LIN {X 0,Y 250.299,Z 339.512,A -85,B 0,C 180,E1 -19332.01,E2 -19332.01} C_VEL
LIN {X 0,Y 247.763,Z 349.944,A -85,B 0,C 180,E1 -19334.367,E2 -19334.367} C_VEL
LIN {X 0,Y 245.729,Z 358.546,A -85,B 0,C 180,E1 -19336.774,E2 -19336.774} C_VEL
LIN {X 0,Y 243.702,Z 366.814,A -85,B 0,C 180,E1 -19339.617,E2 -19339.617} C_VEL
LIN {X 0,Y 242.058,Z 373.465,A -85,B 0,C 180,E1 -19342.493,E2 -19342.493} C_VEL
LIN {X 0,Y 240.854,Z 379.369,A -85,B 0,C 180,E1 -19345.817,E2 -19345.817} C_VEL
LIN {X 0,Y 240.239,Z 382.789,A -85,B 0,C 180,E1 -19348.324,E2 -19348.324} C_VEL
LIN {X 0,Y 239.9,Z 386.062,A -85,B 0,C 180,E1 -19351.679,E2 -19351.679} C_VEL
LIN {X 0,Y 239.798,Z 387.954,A -85,B 0,C 180,E1 -19355.044,E2 -19355.044} C_VEL
LIN {X 0,Y 239.733,Z 388.523,A -85,B 0,C 180,E1 -19358.429,E2 -19358.429} C_VEL
LIN {X 0,Y 239.976,Z 387.764,A -85,B 0,C 180,E1 -19361.83,E2 -19361.83} C_VEL
LIN {X 0,Y 240.849,Z 385.65,A -85,B 0,C 180,E1 -19365.226,E2 -19365.226} C_VEL
LIN {X 0,Y 242.1,Z 382.123,A -85,B 0,C 180,E1 -19368.622,E2 -19368.622} C_VEL
LIN {X 0,Y 244.054,Z 377.068,A -85,B 0,C 180,E1 -19371.985,E2 -19371.985} C_VEL
LIN {X 0,Y 245.959,Z 372.141,A -85,B 0,C 180,E1 -19374.477,E2 -19374.477} C_VEL
LIN {X 0,Y 248.687,Z 365.031,A -85,B 0,C 180,E1 -19377.338,E2 -19377.338} C_VEL
LIN {X 0,Y 251.596,Z 357.106,A -85,B 0,C 180,E1 -19379.879,E2 -19379.879} C_VEL
LIN {X 0,Y 254.542,Z 348.555,A -85,B 0,C 180,E1 -19382.107,E2 -19382.107} C_VEL
LIN {X 0,Y 257.482,Z 339.581,A -85,B 0,C 180,E1 -19384.025,E2 -19384.025} C_VEL
LIN {X 0,Y 260.937,Z 328.34,A -85,B 0,C 180,E1 -19385.962,E2 -19385.962} C_VEL
LIN {X 0,Y 263.827,Z 317.083,A -85,B 0,C 180,E1 -19387.543,E2 -19387.543} C_VEL
LIN {X 0,Y 266.901,Z 304.117,A -85,B 0,C 180,E1 -19388.952,E2 -19388.952} C_VEL
LIN {X 0,Y 269.11,Z 291.695,A -85,B 0,C 180,E1 -19390.024,E2 -19390.024} C_VEL
LIN {X 0,Y 271.038,Z 277.918,A -85,B 0,C 180,E1 -19390.904,E2 -19390.904} C_VEL
LIN {X 0,Y 272.445,Z 263.387,A -85,B 0,C 180,E1 -19391.526,E2 -19391.526} C_VEL
LIN {X 0,Y 276.12,Z 188.093,A -85,B 0,C 180,E1 -19393.435,E2 -19393.435} C_VEL
LIN {X 0,Y 270.633,Z 176.107,A -85,B 0,C 180,E1 -19394.84,E2 -19394.84} C_VEL
LIN {X 0,Y 263.557,Z 162.452,A -85,B 0,C 180,E1 -19396.724,E2 -19396.724} C_VEL
LIN {X 0,Y 256.694,Z 150.677,A -85,B 0,C 180,E1 -19398.658,E2 -19398.658} C_VEL
LIN {X 0,Y 251.055,Z 141.941,A -85,B 0,C 180,E1 -19400.342,E2 -19400.342} C_VEL
LIN {X 0,Y 248.074,Z 137.811,A -85,B 0,C 180,E1 -19401.267,E2 -19401.267} C_VEL
LIN {X 0,Y 245.815,Z 134.692,A -85,B 0,C 180,E1 -19401.993,E2 -19401.993} C_VEL
LIN {X 0,Y 245.019,Z 133.451,A -85,B 0,C 180,E1 -19402.261,E2 -19402.261} C_VEL
LIN {X 0,Y 242.963,Z 131.326,A -85,B 0,C 180,E1 -19402.92,E2 -19402.92} C_VEL
LIN {X 0,Y 242.054,Z 129.048,A -85,B 0,C 180,E1 -19403.278,E2 -19403.278} C_VEL
LIN {X 0,Y 241.967,Z 128.465,A -85,B 0,C 180,E1 -19403.393,E2 -19403.393} C_VEL
LIN {X 0,Y 241.989,Z 128.461,A -85,B 0,C 180,E1 -19407.377,E2 -19407.377} C_VEL
LIN {X 0,Y 241.979,Z 128.46,A -85,B 0,C 180,E1 -19410.612,E2 -19410.612} C_VEL
LIN {X 0,Y 242.034,Z 128.452,A -85,B 0,C 180,E1 -19414.179,E2 -19414.179} C_VEL
LIN {X 0,Y 242.023,Z 128.453,A -85,B 0,C 180,E1 -19418.316,E2 -19418.316} C_VEL
LIN {X 0,Y 242.129,Z 128.446,A -85,B 0,C 180,E1 -19423.306,E2 -19423.306} C_VEL
LIN {X 0,Y 242.18,Z 128.442,A -85,B 0,C 180,E1 -19428.279,E2 -19428.279} C_VEL
LIN {X 0,Y 242.374,Z 128.404,A -85,B 0,C 180,E1 -19431.663,E2 -19431.663} C_VEL
LIN {X 0,Y 242.242,Z 128.426,A -85,B 0,C 180,E1 -19435.007,E2 -19435.007} C_VEL
LIN {X 0,Y 242.434,Z 128.399,A -85,B 0,C 180,E1 -19437.247,E2 -19437.247} C_VEL
LIN {X 0,Y 241.89,Z 128.48,A -85,B 0,C 180,E1 -19438.635,E2 -19438.635} C_VEL
LIN {X 0,Y 240.317,Z 128.675,A -85,B 0,C 180,E1 -19439.998,E2 -19439.998} C_VEL
LIN {X 0,Y 236.438,Z 129.153,A -85,B 0,C 180,E1 -19442.741,E2 -19442.741} C_VEL
LIN {X 0,Y 235.31,Z 129.299,A -85,B 0,C 180,E1 -19444.176,E2 -19444.176} C_VEL
LIN {X 0,Y 235.209,Z 129.302,A -85,B 0,C 180,E1 -19444.663,E2 -19444.663} C_VEL
LIN {X 0,Y 235.356,Z 129.277,A -85,B 0,C 180,E1 -19446.86,E2 -19446.86} C_VEL
LIN {X 0,Y 235.215,Z 129.3,A -85,B 0,C 180,E1 -19450.327,E2 -19450.327} C_VEL
LIN {X 0,Y 235.115,Z 129.308,A -85,B 0,C 180,E1 -19455.606,E2 -19455.606} C_VEL
LIN {X 0,Y 235.01,Z 129.33,A -85,B 0,C 180,E1 -19459.205,E2 -19459.205} C_VEL
LIN {X 0,Y 234.962,Z 129.34,A -85,B 0,C 180,E1 -19462.882,E2 -19462.882} C_VEL
LIN {X 0,Y 234.969,Z 129.338,A -85,B 0,C 180,E1 -19466.657,E2 -19466.657} C_VEL
LIN {X 0,Y 234.924,Z 129.347,A -85,B 0,C 180,E1 -19470.569,E2 -19470.569} C_VEL
LIN {X 0,Y 234.943,Z 129.341,A -85,B 0,C 180,E1 -19474.636,E2 -19474.636} C_VEL
LIN {X 0,Y 234.986,Z 129.449,A -85,B 0,C 180,E1 -19477.815,E2 -19477.815} C_VEL
LIN {X 0,Y 236.809,Z 135.137,A -85,B 0,C 180,E1 -19481.194,E2 -19481.194} C_VEL
LIN {X 0,Y 239.597,Z 139.561,A -85,B 0,C 180,E1 -19482.228,E2 -19482.228} C_VEL
LIN {X 0,Y 241.523,Z 142.398,A -85,B 0,C 180,E1 -19482.904,E2 -19482.904} C_VEL
LIN {X 0,Y 244.741,Z 147.284,A -85,B 0,C 180,E1 -19483.998,E2 -19483.998} C_VEL
LIN {X 0,Y 250.861,Z 157.168,A -85,B 0,C 180,E1 -19485.964,E2 -19485.964} C_VEL
LIN {X 0,Y 258.46,Z 170.887,A -85,B 0,C 180,E1 -19488.242,E2 -19488.242} C_VEL
LIN {X 0,Y 264.628,Z 183.632,A -85,B 0,C 180,E1 -19489.994,E2 -19489.994} C_VEL
LIN {X 0,Y 270.125,Z 196.27,A -85,B 0,C 180,E1 -19491.493,E2 -19491.493} C_VEL
LIN {X 0,Y 270.262,Z 199.468,A -85,B 0,C 180,E1 -19491.628,E2 -19491.628} C_VEL
LIN {X 0,Y 266.512,Z 273.7,A -85,B 0,C 180,E1 -19493.547,E2 -19493.547} C_VEL
LIN {X 0,Y 264.915,Z 288.292,A -85,B 0,C 180,E1 -19494.175,E2 -19494.175} C_VEL
LIN {X 0,Y 262.763,Z 301.669,A -85,B 0,C 180,E1 -19495.014,E2 -19495.014} C_VEL
LIN {X 0,Y 260.057,Z 314.752,A -85,B 0,C 180,E1 -19496.124,E2 -19496.124} C_VEL
LIN {X 0,Y 256.95,Z 327.404,A -85,B 0,C 180,E1 -19497.535,E2 -19497.535} C_VEL
LIN {X 0,Y 253.786,Z 338.75,A -85,B 0,C 180,E1 -19499.145,E2 -19499.145} C_VEL
LIN {X 0,Y 250.411,Z 349.522,A -85,B 0,C 180,E1 -19501.044,E2 -19501.044} C_VEL
LIN {X 0,Y 246.72,Z 360.041,A -85,B 0,C 180,E1 -19503.343,E2 -19503.343} C_VEL
LIN {X 0,Y 243.494,Z 368.736,A -85,B 0,C 180,E1 -19505.713,E2 -19505.713} C_VEL
LIN {X 0,Y 240.238,Z 377.097,A -85,B 0,C 180,E1 -19508.55,E2 -19508.55} C_VEL
LIN {X 0,Y 237.934,Z 382.937,A -85,B 0,C 180,E1 -19511.039,E2 -19511.039} C_VEL
LIN {X 0,Y 235.697,Z 389.202,A -85,B 0,C 180,E1 -19514.433,E2 -19514.433} C_VEL
LIN {X 0,Y 233.997,Z 393.839,A -85,B 0,C 180,E1 -19517.863,E2 -19517.863} C_VEL
LIN {X 0,Y 233.089,Z 397.01,A -85,B 0,C 180,E1 -19521.329,E2 -19521.329} C_VEL
LIN {X 0,Y 232.687,Z 398.825,A -85,B 0,C 180,E1 -19524.801,E2 -19524.801} C_VEL
LIN {X 0,Y 232.713,Z 399.315,A -85,B 0,C 180,E1 -19528.269,E2 -19528.269} C_VEL
LIN {X 0,Y 232.756,Z 399.06,A -85,B 0,C 180,E1 -19530,E2 -19530} C_VEL
LIN {X 0,Y 232.719,Z 398.468,A -85,B 0,C 180,E1 -19531.73,E2 -19531.73} C_VEL
LIN {X 0,Y 232.686,Z 396.257,A -85,B 0,C 180,E1 -19535.198,E2 -19535.198} C_VEL
LIN {X 0,Y 232.999,Z 392.624,A -85,B 0,C 180,E1 -19538.674,E2 -19538.674} C_VEL
LIN {X 0,Y 233.751,Z 387.46,A -85,B 0,C 180,E1 -19542.149,E2 -19542.149} C_VEL
LIN {X 0,Y 234.837,Z 382.452,A -85,B 0,C 180,E1 -19544.737,E2 -19544.737} C_VEL
LIN {X 0,Y 236.45,Z 375.152,A -85,B 0,C 180,E1 -19547.778,E2 -19547.778} C_VEL
LIN {X 0,Y 238.234,Z 367.715,A -85,B 0,C 180,E1 -19550.281,E2 -19550.281} C_VEL
LIN {X 0,Y 240.502,Z 358.652,A -85,B 0,C 180,E1 -19552.78,E2 -19552.78} C_VEL
LIN {X 0,Y 242.794,Z 349.642,A -85,B 0,C 180,E1 -19554.817,E2 -19554.817} C_VEL
LIN {X 0,Y 245.347,Z 338.883,A -85,B 0,C 180,E1 -19556.818,E2 -19556.818} C_VEL
LIN {X 0,Y 247.932,Z 326.71,A -85,B 0,C 180,E1 -19558.643,E2 -19558.643} C_VEL
LIN {X 0,Y 250.264,Z 314.155,A -85,B 0,C 180,E1 -19560.13,E2 -19560.13} C_VEL
LIN {X 0,Y 252.468,Z 300.66,A -85,B 0,C 180,E1 -19561.346,E2 -19561.346} C_VEL
LIN {X 0,Y 254.179,Z 286.6,A -85,B 0,C 180,E1 -19562.275,E2 -19562.275} C_VEL
LIN {X 0,Y 255.333,Z 273.104,A -85,B 0,C 180,E1 -19562.871,E2 -19562.871} C_VEL
LIN {X 0,Y 258.627,Z 191.88,A -85,B 0,C 180,E1 -19565.065,E2 -19565.065} C_VEL
LIN {X 0,Y 256.927,Z 179.947,A -85,B 0,C 180,E1 -19565.694,E2 -19565.694} C_VEL
LIN {X 0,Y 250.007,Z 162.691,A -85,B 0,C 180,E1 -19567.312,E2 -19567.312} C_VEL
LIN {X 0,Y 242.529,Z 146.936,A -85,B 0,C 180,E1 -19569.099,E2 -19569.099} C_VEL
LIN {X 0,Y 237.887,Z 138.311,A -85,B 0,C 180,E1 -19570.243,E2 -19570.243} C_VEL
LIN {X 0,Y 236.625,Z 135.625,A -85,B 0,C 180,E1 -19570.617,E2 -19570.617} C_VEL
LIN {X 0,Y 234.922,Z 129.349,A -85,B 0,C 180,E1 -19573.477,E2 -19573.477} C_VEL
LIN {X 0,Y 234.973,Z 129.337,A -85,B 0,C 180,E1 -19576.534,E2 -19576.534} C_VEL
LIN {X 0,Y 234.954,Z 129.318,A -85,B 0,C 180,E1 -19581.086,E2 -19581.086} C_VEL
LIN {X 0,Y 234.96,Z 129.34,A -85,B 0,C 180,E1 -19585.367,E2 -19585.367} C_VEL
LIN {X 0,Y 234.968,Z 129.336,A -85,B 0,C 180,E1 -19590.157,E2 -19590.157} C_VEL
LIN {X 0,Y 234.993,Z 129.337,A -85,B 0,C 180,E1 -19593.794,E2 -19593.794} C_VEL
LIN {X 0,Y 235.011,Z 129.336,A -85,B 0,C 180,E1 -19598.97,E2 -19598.97} C_VEL
LIN {X 0,Y 235.095,Z 129.322,A -85,B 0,C 180,E1 -19603.06,E2 -19603.06} C_VEL
LIN {X 0,Y 235.118,Z 129.309,A -85,B 0,C 180,E1 -19607.922,E2 -19607.922} C_VEL
LIN {X 0,Y 235.368,Z 129.29,A -85,B 0,C 180,E1 -19611.414,E2 -19611.414} C_VEL
LIN {X 0,Y 235.397,Z 129.278,A -85,B 0,C 180,E1 -19613.141,E2 -19613.141} C_VEL
LIN {X 0,Y 235.595,Z 129.265,A -85,B 0,C 180,E1 -19618.291,E2 -19618.291} C_VEL
LIN {X 0,Y 235.594,Z 129.245,A -85,B 0,C 180,E1 -19621.71,E2 -19621.71} C_VEL
LIN {X 0,Y 235.359,Z 129.29,A -85,B 0,C 180,E1 -19626.86,E2 -19626.86} C_VEL
LIN {X 0,Y 235.214,Z 129.293,A -85,B 0,C 180,E1 -19630.328,E2 -19630.328} C_VEL
LIN {X 0,Y 235.114,Z 129.318,A -85,B 0,C 180,E1 -19635.607,E2 -19635.607} C_VEL
LIN {X 0,Y 235.02,Z 129.325,A -85,B 0,C 180,E1 -19639.205,E2 -19639.205} C_VEL
LIN {X 0,Y 234.981,Z 129.338,A -85,B 0,C 180,E1 -19642.881,E2 -19642.881} C_VEL
LIN {X 0,Y 234.97,Z 129.335,A -85,B 0,C 180,E1 -19646.658,E2 -19646.658} C_VEL
LIN {X 0,Y 234.931,Z 129.338,A -85,B 0,C 180,E1 -19650.568,E2 -19650.568} C_VEL
LIN {X 0,Y 234.93,Z 129.346,A -85,B 0,C 180,E1 -19654.639,E2 -19654.639} C_VEL
LIN {X 0,Y 234.942,Z 129.344,A -85,B 0,C 180,E1 -19658.945,E2 -19658.945} C_VEL
LIN {X 0,Y 234.89,Z 129.351,A -85,B 0,C 180,E1 -19663.486,E2 -19663.486} C_VEL
LIN {X 0,Y 234.891,Z 129.345,A -85,B 0,C 180,E1 -19666.515,E2 -19666.515} C_VEL
LIN {X 0,Y 234.918,Z 129.323,A -85,B 0,C 180,E1 -19671.079,E2 -19671.079} C_VEL
LIN {X 0,Y 234.925,Z 129.482,A -85,B 0,C 180,E1 -19675.242,E2 -19675.242} C_VEL
LIN {X 0,Y 235.997,Z 132.308,A -85,B 0,C 180,E1 -19675.554,E2 -19675.554} C_VEL
LIN {X 0,Y 237.69,Z 134.682,A -85,B 0,C 180,E1 -19675.96,E2 -19675.96} C_VEL
LIN {X 0,Y 245.144,Z 147.089,A -85,B 0,C 180,E1 -19677.728,E2 -19677.728} C_VEL
LIN {X 0,Y 252.479,Z 162.49,A -85,B 0,C 180,E1 -19679.441,E2 -19679.441} C_VEL
LIN {X 0,Y 259.074,Z 178.849,A -85,B 0,C 180,E1 -19680.953,E2 -19680.953} C_VEL
LIN {X 0,Y 255.684,Z 263.548,A -85,B 0,C 180,E1 -19683.25,E2 -19683.25} C_VEL
LIN {X 0,Y 254.601,Z 277.468,A -85,B 0,C 180,E1 -19683.9,E2 -19683.9} C_VEL
LIN {X 0,Y 253.037,Z 291.055,A -85,B 0,C 180,E1 -19684.831,E2 -19684.831} C_VEL
LIN {X 0,Y 251.046,Z 304.269,A -85,B 0,C 180,E1 -19686.051,E2 -19686.051} C_VEL
LIN {X 0,Y 248.647,Z 317.006,A -85,B 0,C 180,E1 -19687.569,E2 -19687.569} C_VEL
LIN {X 0,Y 246.3,Z 328.565,A -85,B 0,C 180,E1 -19689.323,E2 -19689.323} C_VEL
LIN {X 0,Y 243.584,Z 340.14,A -85,B 0,C 180,E1 -19691.496,E2 -19691.496} C_VEL
LIN {X 0,Y 240.965,Z 350.495,A -85,B 0,C 180,E1 -19693.914,E2 -19693.914} C_VEL
LIN {X 0,Y 238.84,Z 359.033,A -85,B 0,C 180,E1 -19696.385,E2 -19696.385} C_VEL
LIN {X 0,Y 236.76,Z 367.23,A -85,B 0,C 180,E1 -19699.309,E2 -19699.309} C_VEL
LIN {X 0,Y 235.049,Z 373.826,A -85,B 0,C 180,E1 -19702.268,E2 -19702.268} C_VEL
LIN {X 0,Y 233.791,Z 379.681,A -85,B 0,C 180,E1 -19705.69,E2 -19705.69} C_VEL
LIN {X 0,Y 233.166,Z 383.079,A -85,B 0,C 180,E1 -19708.273,E2 -19708.273} C_VEL
LIN {X 0,Y 232.808,Z 386.299,A -85,B 0,C 180,E1 -19711.73,E2 -19711.73} C_VEL
LIN {X 0,Y 232.694,Z 388.147,A -85,B 0,C 180,E1 -19715.199,E2 -19715.199} C_VEL
LIN {X 0,Y 232.639,Z 388.678,A -85,B 0,C 180,E1 -19718.688,E2 -19718.688} C_VEL
LIN {X 0,Y 232.954,Z 387.88,A -85,B 0,C 180,E1 -19722.192,E2 -19722.192} C_VEL
LIN {X 0,Y 233.89,Z 385.726,A -85,B 0,C 180,E1 -19725.69,E2 -19725.69} C_VEL
LIN {X 0,Y 235.238,Z 382.159,A -85,B 0,C 180,E1 -19729.186,E2 -19729.186} C_VEL
LIN {X 0,Y 237.338,Z 377.06,A -85,B 0,C 180,E1 -19732.641,E2 -19732.641} C_VEL
LIN {X 0,Y 239.39,Z 372.086,A -85,B 0,C 180,E1 -19735.195,E2 -19735.195} C_VEL
LIN {X 0,Y 242.272,Z 364.924,A -85,B 0,C 180,E1 -19738.125,E2 -19738.125} C_VEL
LIN {X 0,Y 245.476,Z 356.648,A -85,B 0,C 180,E1 -19740.805,E2 -19740.805} C_VEL
LIN {X 0,Y 248.445,Z 348.324,A -85,B 0,C 180,E1 -19742.994,E2 -19742.994} C_VEL
LIN {X 0,Y 252.201,Z 337.302,A -85,B 0,C 180,E1 -19745.327,E2 -19745.327} C_VEL
LIN {X 0,Y 255.677,Z 326.057,A -85,B 0,C 180,E1 -19747.21,E2 -19747.21} C_VEL
LIN {X 0,Y 258.561,Z 315.115,A -85,B 0,C 180,E1 -19748.695,E2 -19748.695} C_VEL
LIN {X 0,Y 261.317,Z 303.419,A -85,B 0,C 180,E1 -19749.949,E2 -19749.949} C_VEL
LIN {X 0,Y 263.655,Z 290.763,A -85,B 0,C 180,E1 -19751.026,E2 -19751.026} C_VEL
LIN {X 0,Y 265.584,Z 276.865,A -85,B 0,C 180,E1 -19751.905,E2 -19751.905} C_VEL
LIN {X 0,Y 266.929,Z 263.262,A -85,B 0,C 180,E1 -19752.473,E2 -19752.473} C_VEL
LIN {X 0,Y 270.633,Z 190.333,A -85,B 0,C 180,E1 -19754.347,E2 -19754.347} C_VEL
LIN {X 0,Y 265.098,Z 178.323,A -85,B 0,C 180,E1 -19755.833,E2 -19755.833} C_VEL
LIN {X 0,Y 257.932,Z 164.518,A -85,B 0,C 180,E1 -19757.845,E2 -19757.845} C_VEL
LIN {X 0,Y 250.491,Z 151.915,A -85,B 0,C 180,E1 -19760.07,E2 -19760.07} C_VEL
LIN {X 0,Y 247.075,Z 146.825,A -85,B 0,C 180,E1 -19761.14,E2 -19761.14} C_VEL
LIN {X 0,Y 244.457,Z 143.159,A -85,B 0,C 180,E1 -19761.986,E2 -19761.986} C_VEL
LIN {X 0,Y 241.366,Z 138.925,A -85,B 0,C 180,E1 -19763.025,E2 -19763.025} C_VEL
LIN {X 0,Y 239.077,Z 135.911,A -85,B 0,C 180,E1 -19763.821,E2 -19763.821} C_VEL
LIN {X 0,Y 238.258,Z 134.511,A -85,B 0,C 180,E1 -19764.128,E2 -19764.128} C_VEL
LIN {X 0,Y 235.996,Z 132.33,A -85,B 0,C 180,E1 -19764.917,E2 -19764.917} C_VEL
LIN {X 0,Y 234.964,Z 129.694,A -85,B 0,C 180,E1 -19765.367,E2 -19765.367} C_VEL
LIN {X 0,Y 234.897,Z 129.352,A -85,B 0,C 180,E1 -19765.462,E2 -19765.462} C_VEL
LIN {X 0,Y 234.901,Z 129.344,A -85,B 0,C 180,E1 -19769.427,E2 -19769.427} C_VEL
LIN {X 0,Y 234.97,Z 129.331,A -85,B 0,C 180,E1 -19773.806,E2 -19773.806} C_VEL
LIN {X 0,Y 234.992,Z 129.334,A -85,B 0,C 180,E1 -19778.968,E2 -19778.968} C_VEL
LIN {X 0,Y 235.065,Z 129.323,A -85,B 0,C 180,E1 -19783.086,E2 -19783.086} C_VEL
LIN {X 0,Y 235.112,Z 129.32,A -85,B 0,C 180,E1 -19787.922,E2 -19787.922} C_VEL
LIN {X 0,Y 235.313,Z 129.282,A -85,B 0,C 180,E1 -19791.411,E2 -19791.411} C_VEL
LIN {X 0,Y 235.353,Z 129.293,A -85,B 0,C 180,E1 -19793.14,E2 -19793.14} C_VEL
LIN {X 0,Y 235.594,Z 129.263,A -85,B 0,C 180,E1 -19798.29,E2 -19798.29} C_VEL
LIN {X 0,Y 235.594,Z 129.247,A -85,B 0,C 180,E1 -19801.709,E2 -19801.709} C_VEL
LIN {X 0,Y 235.209,Z 129.302,A -85,B 0,C 180,E1 -19804.663,E2 -19804.663} C_VEL
LIN {X 0,Y 234.506,Z 129.392,A -85,B 0,C 180,E1 -19806.094,E2 -19806.094} C_VEL
LIN {X 0,Y 231.61,Z 129.759,A -85,B 0,C 180,E1 -19808.428,E2 -19808.428} C_VEL
LIN {X 0,Y 229.176,Z 130.052,A -85,B 0,C 180,E1 -19810.331,E2 -19810.331} C_VEL
LIN {X 0,Y 228.147,Z 130.176,A -85,B 0,C 180,E1 -19811.809,E2 -19811.809} C_VEL
LIN {X 0,Y 228.071,Z 130.188,A -85,B 0,C 180,E1 -19812.31,E2 -19812.31} C_VEL
LIN {X 0,Y 228.059,Z 130.185,A -85,B 0,C 180,E1 -19816.102,E2 -19816.102} C_VEL
LIN {X 0,Y 227.944,Z 130.204,A -85,B 0,C 180,E1 -19819.825,E2 -19819.825} C_VEL
LIN {X 0,Y 227.915,Z 130.213,A -85,B 0,C 180,E1 -19823.632,E2 -19823.632} C_VEL
LIN {X 0,Y 227.88,Z 130.219,A -85,B 0,C 180,E1 -19827.555,E2 -19827.555} C_VEL
LIN {X 0,Y 227.869,Z 130.219,A -85,B 0,C 180,E1 -19831.622,E2 -19831.622} C_VEL
LIN {X 0,Y 227.906,Z 130.334,A -85,B 0,C 180,E1 -19835.867,E2 -19835.867} C_VEL
LIN {X 0,Y 229.35,Z 134.78,A -85,B 0,C 180,E1 -19838.775,E2 -19838.775} C_VEL
LIN {X 0,Y 232.325,Z 139.331,A -85,B 0,C 180,E1 -19839.996,E2 -19839.996} C_VEL
LIN {X 0,Y 233.89,Z 141.41,A -85,B 0,C 180,E1 -19840.597,E2 -19840.597} C_VEL
LIN {X 0,Y 238.409,Z 148.298,A -85,B 0,C 180,E1 -19842.287,E2 -19842.287} C_VEL
LIN {X 0,Y 241.45,Z 153.042,A -85,B 0,C 180,E1 -19843.362,E2 -19843.362} C_VEL
LIN {X 0,Y 247.777,Z 163.591,A -85,B 0,C 180,E1 -19845.473,E2 -19845.473} C_VEL
LIN {X 0,Y 255.055,Z 177.052,A -85,B 0,C 180,E1 -19847.731,E2 -19847.731} C_VEL
LIN {X 0,Y 262.247,Z 192.588,A -85,B 0,C 180,E1 -19849.843,E2 -19849.843} C_VEL
LIN {X 0,Y 264.865,Z 198.903,A -85,B 0,C 180,E1 -19850.589,E2 -19850.589} C_VEL
LIN {X 0,Y 260.984,Z 274.124,A -85,B 0,C 180,E1 -19852.585,E2 -19852.585} C_VEL
LIN {X 0,Y 259.456,Z 287.755,A -85,B 0,C 180,E1 -19853.179,E2 -19853.179} C_VEL
LIN {X 0,Y 257.436,Z 300.106,A -85,B 0,C 180,E1 -19853.938,E2 -19853.938} C_VEL
LIN {X 0,Y 255.086,Z 311.678,A -85,B 0,C 180,E1 -19854.891,E2 -19854.891} C_VEL
LIN {X 0,Y 251.767,Z 324.935,A -85,B 0,C 180,E1 -19856.303,E2 -19856.303} C_VEL
LIN {X 0,Y 248.486,Z 336.606,A -85,B 0,C 180,E1 -19857.919,E2 -19857.919} C_VEL
LIN {X 0,Y 244.923,Z 347.777,A -85,B 0,C 180,E1 -19859.857,E2 -19859.857} C_VEL
LIN {X 0,Y 240.999,Z 358.557,A -85,B 0,C 180,E1 -19862.186,E2 -19862.186} C_VEL
LIN {X 0,Y 237.558,Z 367.473,A -85,B 0,C 180,E1 -19864.597,E2 -19864.597} C_VEL
LIN {X 0,Y 234.054,Z 376.027,A -85,B 0,C 180,E1 -19867.49,E2 -19867.49} C_VEL
LIN {X 0,Y 231.177,Z 382.942,A -85,B 0,C 180,E1 -19870.463,E2 -19870.463} C_VEL
LIN {X 0,Y 228.838,Z 389.169,A -85,B 0,C 180,E1 -19873.954,E2 -19873.954} C_VEL
LIN {X 0,Y 227.005,Z 393.758,A -85,B 0,C 180,E1 -19877.483,E2 -19877.483} C_VEL
LIN {X 0,Y 226.032,Z 396.899,A -85,B 0,C 180,E1 -19881.056,E2 -19881.056} C_VEL
LIN {X 0,Y 225.591,Z 398.684,A -85,B 0,C 180,E1 -19884.637,E2 -19884.637} C_VEL
LIN {X 0,Y 225.609,Z 399.144,A -85,B 0,C 180,E1 -19888.215,E2 -19888.215} C_VEL
LIN {X 0,Y 225.671,Z 398.876,A -85,B 0,C 180,E1 -19890,E2 -19890} C_VEL
LIN {X 0,Y 225.614,Z 398.268,A -85,B 0,C 180,E1 -19891.785,E2 -19891.785} C_VEL
LIN {X 0,Y 225.589,Z 396.026,A -85,B 0,C 180,E1 -19895.362,E2 -19895.362} C_VEL
LIN {X 0,Y 225.953,Z 392.361,A -85,B 0,C 180,E1 -19898.947,E2 -19898.947} C_VEL
LIN {X 0,Y 226.763,Z 387.162,A -85,B 0,C 180,E1 -19902.53,E2 -19902.53} C_VEL
LIN {X 0,Y 227.916,Z 382.117,A -85,B 0,C 180,E1 -19905.195,E2 -19905.195} C_VEL
LIN {X 0,Y 229.347,Z 376.011,A -85,B 0,C 180,E1 -19907.844,E2 -19907.844} C_VEL
LIN {X 0,Y 231.528,Z 367.296,A -85,B 0,C 180,E1 -19910.895,E2 -19910.895} C_VEL
LIN {X 0,Y 233.912,Z 358.181,A -85,B 0,C 180,E1 -19913.459,E2 -19913.459} C_VEL
LIN {X 0,Y 236.776,Z 347.137,A -85,B 0,C 180,E1 -19915.964,E2 -19915.964} C_VEL
LIN {X 0,Y 239.529,Z 335.895,A -85,B 0,C 180,E1 -19917.998,E2 -19917.998} C_VEL
LIN {X 0,Y 242.196,Z 323.443,A -85,B 0,C 180,E1 -19919.797,E2 -19919.797} C_VEL
LIN {X 0,Y 244.61,Z 310.438,A -85,B 0,C 180,E1 -19921.262,E2 -19921.262} C_VEL
LIN {X 0,Y 246.763,Z 297.008,A -85,B 0,C 180,E1 -19922.397,E2 -19922.397} C_VEL
LIN {X 0,Y 248.457,Z 282.308,A -85,B 0,C 180,E1 -19923.294,E2 -19923.294} C_VEL
LIN {X 0,Y 249.561,Z 267.663,A -85,B 0,C 180,E1 -19923.853,E2 -19923.853} C_VEL
LIN {X 0,Y 252.574,Z 192.478,A -85,B 0,C 180,E1 -19925.916,E2 -19925.916} C_VEL
LIN {X 0,Y 251.202,Z 182.591,A -85,B 0,C 180,E1 -19926.452,E2 -19926.452} C_VEL
LIN {X 0,Y 245.006,Z 166.927,A -85,B 0,C 180,E1 -19927.97,E2 -19927.97} C_VEL
LIN {X 0,Y 237.942,Z 151.736,A -85,B 0,C 180,E1 -19929.734,E2 -19929.734} C_VEL
LIN {X 0,Y 231.564,Z 139.734,A -85,B 0,C 180,E1 -19931.392,E2 -19931.392} C_VEL
LIN {X 0,Y 229.282,Z 135.378,A -85,B 0,C 180,E1 -19932.077,E2 -19932.077} C_VEL
LIN {X 0,Y 227.848,Z 130.226,A -85,B 0,C 180,E1 -19934.575,E2 -19934.575} C_VEL
LIN {X 0,Y 227.916,Z 130.219,A -85,B 0,C 180,E1 -19937.736,E2 -19937.736} C_VEL
LIN {X 0,Y 227.87,Z 130.201,A -85,B 0,C 180,E1 -19941.914,E2 -19941.914} C_VEL
LIN {X 0,Y 227.889,Z 130.215,A -85,B 0,C 180,E1 -19946.373,E2 -19946.373} C_VEL
LIN {X 0,Y 227.918,Z 130.213,A -85,B 0,C 180,E1 -19950.438,E2 -19950.438} C_VEL
LIN {X 0,Y 227.928,Z 130.216,A -85,B 0,C 180,E1 -19954.426,E2 -19954.426} C_VEL
LIN {X 0,Y 227.961,Z 130.213,A -85,B 0,C 180,E1 -19958.287,E2 -19958.287} C_VEL
LIN {X 0,Y 228.034,Z 130.199,A -85,B 0,C 180,E1 -19962.826,E2 -19962.826} C_VEL
LIN {X 0,Y 228.074,Z 130.185,A -85,B 0,C 180,E1 -19967.544,E2 -19967.544} C_VEL
LIN {X 0,Y 228.298,Z 130.172,A -85,B 0,C 180,E1 -19971.146,E2 -19971.146} C_VEL
LIN {X 0,Y 228.348,Z 130.157,A -85,B 0,C 180,E1 -19972.929,E2 -19972.929} C_VEL
LIN {X 0,Y 228.553,Z 130.142,A -85,B 0,C 180,E1 -19978.238,E2 -19978.238} C_VEL
LIN {X 0,Y 228.552,Z 130.12,A -85,B 0,C 180,E1 -19981.762,E2 -19981.762} C_VEL
LIN {X 0,Y 228.311,Z 130.168,A -85,B 0,C 180,E1 -19987.073,E2 -19987.073} C_VEL
LIN {X 0,Y 228.145,Z 130.173,A -85,B 0,C 180,E1 -19990.652,E2 -19990.652} C_VEL
LIN {X 0,Y 228.065,Z 130.2,A -85,B 0,C 180,E1 -19994.272,E2 -19994.272} C_VEL
LIN {X 0,Y 228.007,Z 130.191,A -85,B 0,C 180,E1 -19997.953,E2 -19997.953} C_VEL
LIN {X 0,Y 227.961,Z 130.212,A -85,B 0,C 180,E1 -20002.348,E2 -20002.348} C_VEL
LIN {X 0,Y 227.943,Z 130.21,A -85,B 0,C 180,E1 -20006.603,E2 -20006.603} C_VEL
LIN {X 0,Y 227.908,Z 130.214,A -85,B 0,C 180,E1 -20010.296,E2 -20010.296} C_VEL
LIN {X 0,Y 227.877,Z 130.225,A -85,B 0,C 180,E1 -20013.721,E2 -20013.721} C_VEL
LIN {X 0,Y 227.844,Z 130.223,A -85,B 0,C 180,E1 -20018.092,E2 -20018.092} C_VEL
LIN {X 0,Y 227.813,Z 130.226,A -85,B 0,C 180,E1 -20022.743,E2 -20022.743} C_VEL
LIN {X 0,Y 227.814,Z 130.232,A -85,B 0,C 180,E1 -20027.259,E2 -20027.259} C_VEL
LIN {X 0,Y 227.844,Z 130.205,A -85,B 0,C 180,E1 -20031.909,E2 -20031.909} C_VEL
LIN {X 0,Y 227.898,Z 130.225,A -85,B 0,C 180,E1 -20033.861,E2 -20033.861} C_VEL
LIN {X 0,Y 228.784,Z 132.881,A -85,B 0,C 180,E1 -20034.155,E2 -20034.155} C_VEL
LIN {X 0,Y 230.553,Z 135.256,A -85,B 0,C 180,E1 -20034.608,E2 -20034.608} C_VEL
LIN {X 0,Y 240.064,Z 150.916,A -85,B 0,C 180,E1 -20036.99,E2 -20036.99} C_VEL
LIN {X 0,Y 247.48,Z 166.738,A -85,B 0,C 180,E1 -20038.801,E2 -20038.801} C_VEL
LIN {X 0,Y 253.012,Z 180.561,A -85,B 0,C 180,E1 -20040.127,E2 -20040.127} C_VEL
LIN {X 0,Y 249.589,Z 263.601,A -85,B 0,C 180,E1 -20042.429,E2 -20042.429} C_VEL
LIN {X 0,Y 248.461,Z 277.568,A -85,B 0,C 180,E1 -20043.091,E2 -20043.091} C_VEL
LIN {X 0,Y 246.852,Z 291.169,A -85,B 0,C 180,E1 -20044.041,E2 -20044.041} C_VEL
LIN {X 0,Y 244.935,Z 303.517,A -85,B 0,C 180,E1 -20045.188,E2 -20045.188} C_VEL
LIN {X 0,Y 242.441,Z 316.431,A -85,B 0,C 180,E1 -20046.736,E2 -20046.736} C_VEL
LIN {X 0,Y 239.96,Z 328.123,A -85,B 0,C 180,E1 -20048.525,E2 -20048.525} C_VEL
LIN {X 0,Y 237.399,Z 338.829,A -85,B 0,C 180,E1 -20050.547,E2 -20050.547} C_VEL
LIN {X 0,Y 234.607,Z 349.429,A -85,B 0,C 180,E1 -20053.018,E2 -20053.018} C_VEL
LIN {X 0,Y 232.39,Z 358.04,A -85,B 0,C 180,E1 -20055.508,E2 -20055.508} C_VEL
LIN {X 0,Y 230.434,Z 365.456,A -85,B 0,C 180,E1 -20058.12,E2 -20058.12} C_VEL
LIN {X 0,Y 228.488,Z 372.436,A -85,B 0,C 180,E1 -20061.153,E2 -20061.153} C_VEL
LIN {X 0,Y 226.936,Z 378.707,A -85,B 0,C 180,E1 -20064.669,E2 -20064.669} C_VEL
LIN {X 0,Y 226.095,Z 383.361,A -85,B 0,C 180,E1 -20068.219,E2 -20068.219} C_VEL
LIN {X 0,Y 225.717,Z 386.529,A -85,B 0,C 180,E1 -20071.785,E2 -20071.785} C_VEL
LIN {X 0,Y 225.581,Z 388.339,A -85,B 0,C 180,E1 -20075.363,E2 -20075.363} C_VEL
LIN {X 0,Y 225.565,Z 388.832,A -85,B 0,C 180,E1 -20078.963,E2 -20078.963} C_VEL
LIN {X 0,Y 225.946,Z 387.996,A -85,B 0,C 180,E1 -20082.576,E2 -20082.576} C_VEL
LIN {X 0,Y 226.985,Z 385.716,A -85,B 0,C 180,E1 -20086.292,E2 -20086.292} C_VEL
LIN {X 0,Y 228.413,Z 382.195,A -85,B 0,C 180,E1 -20089.783,E2 -20089.783} C_VEL
LIN {X 0,Y 230.663,Z 377.052,A -85,B 0,C 180,E1 -20093.334,E2 -20093.334} C_VEL
LIN {X 0,Y 232.838,Z 372.031,A -85,B 0,C 180,E1 -20095.956,E2 -20095.956} C_VEL
LIN {X 0,Y 235.934,Z 364.818,A -85,B 0,C 180,E1 -20098.951,E2 -20098.951} C_VEL
LIN {X 0,Y 239.515,Z 355.863,A -85,B 0,C 180,E1 -20101.882,E2 -20101.882} C_VEL
LIN {X 0,Y 243.022,Z 346.416,A -85,B 0,C 180,E1 -20104.328,E2 -20104.328} C_VEL
LIN {X 0,Y 246.711,Z 335.92,A -85,B 0,C 180,E1 -20106.489,E2 -20106.489} C_VEL
LIN {X 0,Y 249.935,Z 325.603,A -85,B 0,C 180,E1 -20108.216,E2 -20108.216} C_VEL
LIN {X 0,Y 253.004,Z 314.563,A -85,B 0,C 180,E1 -20109.71,E2 -20109.71} C_VEL
LIN {X 0,Y 256.004,Z 301.712,A -85,B 0,C 180,E1 -20111.083,E2 -20111.083} C_VEL
LIN {X 0,Y 258.474,Z 288.461,A -85,B 0,C 180,E1 -20112.165,E2 -20112.165} C_VEL
LIN {X 0,Y 260.299,Z 275.405,A -85,B 0,C 180,E1 -20112.95,E2 -20112.95} C_VEL
LIN {X 0,Y 261.623,Z 261.198,A -85,B 0,C 180,E1 -20113.518,E2 -20113.518} C_VEL
LIN {X 0,Y 265.179,Z 192.496,A -85,B 0,C 180,E1 -20115.307,E2 -20115.307} C_VEL
LIN {X 0,Y 258.449,Z 178.165,A -85,B 0,C 180,E1 -20117.211,E2 -20117.211} C_VEL
LIN {X 0,Y 250.95,Z 164.156,A -85,B 0,C 180,E1 -20119.458,E2 -20119.458} C_VEL
LIN {X 0,Y 244.173,Z 153.052,A -85,B 0,C 180,E1 -20121.63,E2 -20121.63} C_VEL
LIN {X 0,Y 240.127,Z 147.515,A -85,B 0,C 180,E1 -20122.985,E2 -20122.985} C_VEL
LIN {X 0,Y 237.876,Z 144.376,A -85,B 0,C 180,E1 -20123.779,E2 -20123.779} C_VEL
LIN {X 0,Y 235.405,Z 140.805,A -85,B 0,C 180,E1 -20124.691,E2 -20124.691} C_VEL
LIN {X 0,Y 232.56,Z 137.535,A -85,B 0,C 180,E1 -20125.746,E2 -20125.746} C_VEL
LIN {X 0,Y 231.475,Z 135.544,A -85,B 0,C 180,E1 -20126.2,E2 -20126.2} C_VEL
LIN {X 0,Y 229.167,Z 133.463,A -85,B 0,C 180,E1 -20127.085,E2 -20127.085} C_VEL
LIN {X 0,Y 228.021,Z 130.897,A -85,B 0,C 180,E1 -20127.62,E2 -20127.62} C_VEL
LIN {X 0,Y 227.892,Z 130.218,A -85,B 0,C 180,E1 -20127.73,E2 -20127.73} C_VEL
LIN {X 0,Y 227.857,Z 130.224,A -85,B 0,C 180,E1 -20132.441,E2 -20132.441} C_VEL
LIN {X 0,Y 227.896,Z 130.217,A -85,B 0,C 180,E1 -20136.365,E2 -20136.365} C_VEL
LIN {X 0,Y 227.928,Z 130.216,A -85,B 0,C 180,E1 -20140.173,E2 -20140.173} C_VEL
LIN {X 0,Y 228.031,Z 130.206,A -85,B 0,C 180,E1 -20143.896,E2 -20143.896} C_VEL
LIN {X 0,Y 228.068,Z 130.192,A -85,B 0,C 180,E1 -20147.543,E2 -20147.543} C_VEL
LIN {X 0,Y 228.255,Z 130.161,A -85,B 0,C 180,E1 -20151.144,E2 -20151.144} C_VEL
LIN {X 0,Y 228.305,Z 130.167,A -85,B 0,C 180,E1 -20152.927,E2 -20152.927} C_VEL
LIN {X 0,Y 228.552,Z 130.139,A -85,B 0,C 180,E1 -20158.238,E2 -20158.238} C_VEL
LIN {X 0,Y 228.552,Z 130.124,A -85,B 0,C 180,E1 -20161.762,E2 -20161.762} C_VEL
LIN {X 0,Y 228.308,Z 130.156,A -85,B 0,C 180,E1 -20167.073,E2 -20167.073} C_VEL
LIN {X 0,Y 228.147,Z 130.178,A -85,B 0,C 180,E1 -20170.651,E2 -20170.651} C_VEL
LIN {X 0,Y 228.071,Z 130.188,A -85,B 0,C 180,E1 -20172.31,E2 -20172.31} C_VEL
LIN {X 0,Y 227.4,Z 130.285,A -85,B 0,C 180,E1 -20173.785,E2 -20173.785} C_VEL
LIN {X 0,Y 224.471,Z 130.646,A -85,B 0,C 180,E1 -20176.189,E2 -20176.189} C_VEL
LIN {X 0,Y 221.99,Z 130.955,A -85,B 0,C 180,E1 -20178.151,E2 -20178.151} C_VEL
LIN {X 0,Y 220.952,Z 131.076,A -85,B 0,C 180,E1 -20179.677,E2 -20179.677} C_VEL
LIN {X 0,Y 220.882,Z 131.08,A -85,B 0,C 180,E1 -20180.195,E2 -20180.195} C_VEL
LIN {X 0,Y 220.868,Z 131.084,A -85,B 0,C 180,E1 -20184.435,E2 -20184.435} C_VEL
LIN {X 0,Y 220.828,Z 131.091,A -85,B 0,C 180,E1 -20188.514,E2 -20188.514} C_VEL
LIN {X 0,Y 220.82,Z 131.095,A -85,B 0,C 180,E1 -20192.755,E2 -20192.755} C_VEL
LIN {X 0,Y 220.871,Z 131.294,A -85,B 0,C 180,E1 -20193.75,E2 -20193.75} C_VEL
LIN {X 0,Y 221.98,Z 134.501,A -85,B 0,C 180,E1 -20196.064,E2 -20196.064} C_VEL
LIN {X 0,Y 224.217,Z 138.057,A -85,B 0,C 180,E1 -20197.119,E2 -20197.119} C_VEL
LIN {X 0,Y 226.775,Z 141.379,A -85,B 0,C 180,E1 -20198.228,E2 -20198.228} C_VEL
LIN {X 0,Y 230.902,Z 147.444,A -85,B 0,C 180,E1 -20199.941,E2 -20199.941} C_VEL
LIN {X 0,Y 237.021,Z 156.731,A -85,B 0,C 180,E1 -20202.275,E2 -20202.275} C_VEL
LIN {X 0,Y 244.87,Z 170.14,A -85,B 0,C 180,E1 -20205.016,E2 -20205.016} C_VEL
LIN {X 0,Y 252.6,Z 185.272,A -85,B 0,C 180,E1 -20207.501,E2 -20207.501} C_VEL
LIN {X 0,Y 259.397,Z 200.833,A -85,B 0,C 180,E1 -20209.566,E2 -20209.566} C_VEL
LIN {X 0,Y 259.501,Z 203.196,A -85,B 0,C 180,E1 -20209.675,E2 -20209.675} C_VEL
LIN {X 0,Y 255.649,Z 273.413,A -85,B 0,C 180,E1 -20211.539,E2 -20211.539} C_VEL
LIN {X 0,Y 254.078,Z 287.227,A -85,B 0,C 180,E1 -20212.141,E2 -20212.141} C_VEL
LIN {X 0,Y 251.758,Z 300.797,A -85,B 0,C 180,E1 -20212.991,E2 -20212.991} C_VEL
LIN {X 0,Y 249.332,Z 312.233,A -85,B 0,C 180,E1 -20213.955,E2 -20213.955} C_VEL
LIN {X 0,Y 245.914,Z 325.312,A -85,B 0,C 180,E1 -20215.388,E2 -20215.388} C_VEL
LIN {X 0,Y 242.171,Z 337.877,A -85,B 0,C 180,E1 -20217.187,E2 -20217.187} C_VEL
LIN {X 0,Y 238.816,Z 347.982,A -85,B 0,C 180,E1 -20219.002,E2 -20219.002} C_VEL
LIN {X 0,Y 234.749,Z 358.7,A -85,B 0,C 180,E1 -20221.379,E2 -20221.379} C_VEL
LIN {X 0,Y 231.159,Z 367.564,A -85,B 0,C 180,E1 -20223.842,E2 -20223.842} C_VEL
LIN {X 0,Y 227.48,Z 376.071,A -85,B 0,C 180,E1 -20226.802,E2 -20226.802} C_VEL
LIN {X 0,Y 224.29,Z 383.362,A -85,B 0,C 180,E1 -20230.056,E2 -20230.056} C_VEL
LIN {X 0,Y 221.974,Z 389.13,A -85,B 0,C 180,E1 -20233.444,E2 -20233.444} C_VEL
LIN {X 0,Y 220.028,Z 393.677,A -85,B 0,C 180,E1 -20237.08,E2 -20237.08} C_VEL
LIN {X 0,Y 218.995,Z 396.788,A -85,B 0,C 180,E1 -20240.766,E2 -20240.766} C_VEL
LIN {X 0,Y 218.502,Z 398.543,A -85,B 0,C 180,E1 -20244.462,E2 -20244.462} C_VEL
LIN {X 0,Y 218.509,Z 398.974,A -85,B 0,C 180,E1 -20248.157,E2 -20248.157} C_VEL
LIN {X 0,Y 218.587,Z 398.691,A -85,B 0,C 180,E1 -20250,E2 -20250} C_VEL
LIN {X 0,Y 218.513,Z 398.068,A -85,B 0,C 180,E1 -20251.843,E2 -20251.843} C_VEL
LIN {X 0,Y 218.499,Z 395.795,A -85,B 0,C 180,E1 -20255.537,E2 -20255.537} C_VEL
LIN {X 0,Y 218.922,Z 392.099,A -85,B 0,C 180,E1 -20259.236,E2 -20259.236} C_VEL
LIN {X 0,Y 219.785,Z 386.864,A -85,B 0,C 180,E1 -20262.934,E2 -20262.934} C_VEL
LIN {X 0,Y 221.015,Z 381.783,A -85,B 0,C 180,E1 -20265.681,E2 -20265.681} C_VEL
LIN {X 0,Y 222.495,Z 375.635,A -85,B 0,C 180,E1 -20268.413,E2 -20268.413} C_VEL
LIN {X 0,Y 224.847,Z 366.877,A -85,B 0,C 180,E1 -20271.547,E2 -20271.547} C_VEL
LIN {X 0,Y 227.337,Z 357.71,A -85,B 0,C 180,E1 -20274.18,E2 -20274.18} C_VEL
LIN {X 0,Y 230.389,Z 346.603,A -85,B 0,C 180,E1 -20276.74,E2 -20276.74} C_VEL
LIN {X 0,Y 233.242,Z 335.257,A -85,B 0,C 180,E1 -20278.823,E2 -20278.823} C_VEL
LIN {X 0,Y 236.017,Z 322.685,A -85,B 0,C 180,E1 -20280.659,E2 -20280.659} C_VEL
LIN {X 0,Y 238.547,Z 309.53,A -85,B 0,C 180,E1 -20282.151,E2 -20282.151} C_VEL
LIN {X 0,Y 240.772,Z 295.869,A -85,B 0,C 180,E1 -20283.307,E2 -20283.307} C_VEL
LIN {X 0,Y 242.442,Z 281.693,A -85,B 0,C 180,E1 -20284.17,E2 -20284.17} C_VEL
LIN {X 0,Y 243.569,Z 266.724,A -85,B 0,C 180,E1 -20284.741,E2 -20284.741} C_VEL
LIN {X 0,Y 246.658,Z 193.704,A -85,B 0,C 180,E1 -20286.774,E2 -20286.774} C_VEL
LIN {X 0,Y 245.368,Z 184.743,A -85,B 0,C 180,E1 -20287.288,E2 -20287.288} C_VEL
LIN {X 0,Y 239.14,Z 169.095,A -85,B 0,C 180,E1 -20288.885,E2 -20288.885} C_VEL
LIN {X 0,Y 231.701,Z 153.006,A -85,B 0,C 180,E1 -20290.852,E2 -20290.852} C_VEL
LIN {X 0,Y 226.323,Z 143.24,A -85,B 0,C 180,E1 -20292.314,E2 -20292.314} C_VEL
LIN {X 0,Y 223.228,Z 137.829,A -85,B 0,C 180,E1 -20293.193,E2 -20293.193} C_VEL
LIN {X 0,Y 221.968,Z 135.244,A -85,B 0,C 180,E1 -20293.606,E2 -20293.606} C_VEL
LIN {X 0,Y 220.825,Z 131.104,A -85,B 0,C 180,E1 -20295.765,E2 -20295.765} C_VEL
LIN {X 0,Y 220.855,Z 131.08,A -85,B 0,C 180,E1 -20299.793,E2 -20299.793} C_VEL
LIN {X 0,Y 220.833,Z 131.084,A -85,B 0,C 180,E1 -20302.795,E2 -20302.795} C_VEL
LIN {X 0,Y 220.823,Z 131.096,A -85,B 0,C 180,E1 -20307.245,E2 -20307.245} C_VEL
LIN {X 0,Y 220.836,Z 131.095,A -85,B 0,C 180,E1 -20311.487,E2 -20311.487} C_VEL
LIN {X 0,Y 220.867,Z 131.087,A -85,B 0,C 180,E1 -20315.565,E2 -20315.565} C_VEL
LIN {X 0,Y 220.892,Z 131.091,A -85,B 0,C 180,E1 -20319.514,E2 -20319.514} C_VEL
LIN {X 0,Y 221.016,Z 131.078,A -85,B 0,C 180,E1 -20323.37,E2 -20323.37} C_VEL
LIN {X 0,Y 221.106,Z 131.06,A -85,B 0,C 180,E1 -20329.006,E2 -20329.006} C_VEL
LIN {X 0,Y 221.283,Z 131.038,A -85,B 0,C 180,E1 -20332.702,E2 -20332.702} C_VEL
LIN {X 0,Y 221.511,Z 131.019,A -85,B 0,C 180,E1 -20338.182,E2 -20338.182} C_VEL
LIN {X 0,Y 221.51,Z 130.996,A -85,B 0,C 180,E1 -20341.818,E2 -20341.818} C_VEL
LIN {X 0,Y 221.248,Z 131.048,A -85,B 0,C 180,E1 -20347.3,E2 -20347.3} C_VEL
LIN {X 0,Y 221.067,Z 131.056,A -85,B 0,C 180,E1 -20350.997,E2 -20350.997} C_VEL
LIN {X 0,Y 220.996,Z 131.08,A -85,B 0,C 180,E1 -20354.739,E2 -20354.739} C_VEL
LIN {X 0,Y 220.927,Z 131.074,A -85,B 0,C 180,E1 -20358.549,E2 -20358.549} C_VEL
LIN {X 0,Y 220.921,Z 131.089,A -85,B 0,C 180,E1 -20362.698,E2 -20362.698} C_VEL
LIN {X 0,Y 220.886,Z 131.09,A -85,B 0,C 180,E1 -20367.016,E2 -20367.016} C_VEL
LIN {X 0,Y 220.838,Z 131.09,A -85,B 0,C 180,E1 -20370.768,E2 -20370.768} C_VEL
LIN {X 0,Y 220.801,Z 131.106,A -85,B 0,C 180,E1 -20374.955,E2 -20374.955} C_VEL
LIN {X 0,Y 220.807,Z 131.106,A -85,B 0,C 180,E1 -20379.537,E2 -20379.537} C_VEL
LIN {X 0,Y 220.776,Z 131.109,A -85,B 0,C 180,E1 -20384.454,E2 -20384.454} C_VEL
LIN {X 0,Y 220.772,Z 131.111,A -85,B 0,C 180,E1 -20388.048,E2 -20388.048} C_VEL
LIN {X 0,Y 220.817,Z 131.083,A -85,B 0,C 180,E1 -20392.332,E2 -20392.332} C_VEL
LIN {X 0,Y 221.891,Z 134.061,A -85,B 0,C 180,E1 -20392.731,E2 -20392.731} C_VEL
LIN {X 0,Y 223.727,Z 136.397,A -85,B 0,C 180,E1 -20393.232,E2 -20393.232} C_VEL
LIN {X 0,Y 233.331,Z 151.924,A -85,B 0,C 180,E1 -20395.794,E2 -20395.794} C_VEL
LIN {X 0,Y 237.019,Z 158.901,A -85,B 0,C 180,E1 -20396.74,E2 -20396.74} C_VEL
LIN {X 0,Y 244.135,Z 174.928,A -85,B 0,C 180,E1 -20398.544,E2 -20398.544} C_VEL
LIN {X 0,Y 247.055,Z 182.395,A -85,B 0,C 180,E1 -20399.274,E2 -20399.274} C_VEL
LIN {X 0,Y 243.55,Z 263.635,A -85,B 0,C 180,E1 -20401.567,E2 -20401.567} C_VEL
LIN {X 0,Y 242.387,Z 277.657,A -85,B 0,C 180,E1 -20402.243,E2 -20402.243} C_VEL
LIN {X 0,Y 240.718,Z 291.278,A -85,B 0,C 180,E1 -20403.211,E2 -20403.211} C_VEL
LIN {X 0,Y 238.558,Z 304.518,A -85,B 0,C 180,E1 -20404.478,E2 -20404.478} C_VEL
LIN {X 0,Y 235.985,Z 317.271,A -85,B 0,C 180,E1 -20406.061,E2 -20406.061} C_VEL
LIN {X 0,Y 233.421,Z 328.842,A -85,B 0,C 180,E1 -20407.892,E2 -20407.892} C_VEL
LIN {X 0,Y 230.74,Z 339.457,A -85,B 0,C 180,E1 -20409.961,E2 -20409.961} C_VEL
LIN {X 0,Y 227.846,Z 349.98,A -85,B 0,C 180,E1 -20412.498,E2 -20412.498} C_VEL
LIN {X 0,Y 225.459,Z 358.793,A -85,B 0,C 180,E1 -20415.144,E2 -20415.144} C_VEL
LIN {X 0,Y 223.199,Z 366.993,A -85,B 0,C 180,E1 -20418.19,E2 -20418.19} C_VEL
LIN {X 0,Y 221.511,Z 372.813,A -85,B 0,C 180,E1 -20420.873,E2 -20420.873} C_VEL
LIN {X 0,Y 219.898,Z 379.039,A -85,B 0,C 180,E1 -20424.498,E2 -20424.498} C_VEL
LIN {X 0,Y 219.026,Z 383.635,A -85,B 0,C 180,E1 -20428.162,E2 -20428.162} C_VEL
LIN {X 0,Y 218.61,Z 386.76,A -85,B 0,C 180,E1 -20431.843,E2 -20431.843} C_VEL
LIN {X 0,Y 218.483,Z 388.531,A -85,B 0,C 180,E1 -20435.538,E2 -20435.538} C_VEL
LIN {X 0,Y 218.475,Z 388.987,A -85,B 0,C 180,E1 -20439.256,E2 -20439.256} C_VEL
LIN {X 0,Y 218.92,Z 388.112,A -85,B 0,C 180,E1 -20442.987,E2 -20442.987} C_VEL
LIN {X 0,Y 220.017,Z 385.881,A -85,B 0,C 180,E1 -20446.708,E2 -20446.708} C_VEL
LIN {X 0,Y 221.635,Z 382.231,A -85,B 0,C 180,E1 -20450.415,E2 -20450.415} C_VEL
LIN {X 0,Y 224.032,Z 377.043,A -85,B 0,C 180,E1 -20454.068,E2 -20454.068} C_VEL
LIN {X 0,Y 226.33,Z 371.976,A -85,B 0,C 180,E1 -20456.76,E2 -20456.76} C_VEL
LIN {X 0,Y 229.639,Z 364.712,A -85,B 0,C 180,E1 -20459.823,E2 -20459.823} C_VEL
LIN {X 0,Y 232.796,Z 357.177,A -85,B 0,C 180,E1 -20462.363,E2 -20462.363} C_VEL
LIN {X 0,Y 236.442,Z 347.865,A -85,B 0,C 180,E1 -20464.903,E2 -20464.903} C_VEL
LIN {X 0,Y 240.204,Z 337.674,A -85,B 0,C 180,E1 -20467.118,E2 -20467.118} C_VEL
LIN {X 0,Y 243.852,Z 326.753,A -85,B 0,C 180,E1 -20469.016,E2 -20469.016} C_VEL
LIN {X 0,Y 247.093,Z 315.515,A -85,B 0,C 180,E1 -20470.589,E2 -20470.589} C_VEL
LIN {X 0,Y 250,Z 303.834,A -85,B 0,C 180,E1 -20471.887,E2 -20471.887} C_VEL
LIN {X 0,Y 252.776,Z 290.015,A -85,B 0,C 180,E1 -20473.072,E2 -20473.072} C_VEL
LIN {X 0,Y 254.775,Z 276.424,A -85,B 0,C 180,E1 -20473.924,E2 -20473.924} C_VEL
LIN {X 0,Y 256.184,Z 262.332,A -85,B 0,C 180,E1 -20474.51,E2 -20474.51} C_VEL
LIN {X 0,Y 259.907,Z 195.057,A -85,B 0,C 180,E1 -20476.272,E2 -20476.272} C_VEL
LIN {X 0,Y 253.026,Z 180.416,A -85,B 0,C 180,E1 -20478.322,E2 -20478.322} C_VEL
LIN {X 0,Y 245.566,Z 166.471,A -85,B 0,C 180,E1 -20480.691,E2 -20480.691} C_VEL
LIN {X 0,Y 240.151,Z 157.761,A -85,B 0,C 180,E1 -20482.514,E2 -20482.514} C_VEL
LIN {X 0,Y 234.653,Z 150.05,A -85,B 0,C 180,E1 -20484.476,E2 -20484.476} C_VEL
LIN {X 0,Y 231.583,Z 145.868,A -85,B 0,C 180,E1 -20485.645,E2 -20485.645} C_VEL
LIN {X 0,Y 228.939,Z 142.302,A -85,B 0,C 180,E1 -20486.702,E2 -20486.702} C_VEL
LIN {X 0,Y 227.684,Z 140.914,A -85,B 0,C 180,E1 -20487.206,E2 -20487.206} C_VEL
LIN {X 0,Y 225.5,Z 138.051,A -85,B 0,C 180,E1 -20488.137,E2 -20488.137} C_VEL
LIN {X 0,Y 224.654,Z 136.564,A -85,B 0,C 180,E1 -20488.53,E2 -20488.53} C_VEL
LIN {X 0,Y 222.244,Z 134.553,A -85,B 0,C 180,E1 -20489.558,E2 -20489.558} C_VEL
LIN {X 0,Y 220.992,Z 131.959,A -85,B 0,C 180,E1 -20490.204,E2 -20490.204} C_VEL
LIN {X 0,Y 220.85,Z 131.091,A -85,B 0,C 180,E1 -20490.38,E2 -20490.38} C_VEL
LIN {X 0,Y 220.877,Z 131.086,A -85,B 0,C 180,E1 -20493.547,E2 -20493.547} C_VEL
LIN {X 0,Y 220.868,Z 131.085,A -85,B 0,C 180,E1 -20497.552,E2 -20497.552} C_VEL
LIN {X 0,Y 220.965,Z 131.074,A -85,B 0,C 180,E1 -20502.589,E2 -20502.589} C_VEL
LIN {X 0,Y 221.006,Z 131.068,A -85,B 0,C 180,E1 -20507.138,E2 -20507.138} C_VEL
LIN {X 0,Y 221.196,Z 131.04,A -85,B 0,C 180,E1 -20510.859,E2 -20510.859} C_VEL
LIN {X 0,Y 221.125,Z 131.061,A -85,B 0,C 180,E1 -20514.528,E2 -20514.528} C_VEL
LIN {X 0,Y 221.51,Z 131.016,A -85,B 0,C 180,E1 -20518.182,E2 -20518.182} C_VEL
LIN {X 0,Y 221.51,Z 131.002,A -85,B 0,C 180,E1 -20521.818,E2 -20521.818} C_VEL
LIN {X 0,Y 221.246,Z 131.037,A -85,B 0,C 180,E1 -20527.3,E2 -20527.3} C_VEL
LIN {X 0,Y 221.069,Z 131.057,A -85,B 0,C 180,E1 -20530.996,E2 -20530.996} C_VEL
LIN {X 0,Y 220.997,Z 131.074,A -85,B 0,C 180,E1 -20534.738,E2 -20534.738} C_VEL
LIN {X 0,Y 220.924,Z 131.089,A -85,B 0,C 180,E1 -20538.549,E2 -20538.549} C_VEL
LIN {X 0,Y 220.882,Z 131.08,A -85,B 0,C 180,E1 -20540.195,E2 -20540.195} C_VEL
LIN {X 0,Y 220.255,Z 131.164,A -85,B 0,C 180,E1 -20541.717,E2 -20541.717} C_VEL
LIN {X 0,Y 217.415,Z 131.518,A -85,B 0,C 180,E1 -20544.201,E2 -20544.201} C_VEL
LIN {X 0,Y 214.117,Z 131.936,A -85,B 0,C 180,E1 -20547.273,E2 -20547.273} C_VEL
LIN {X 0,Y 213.766,Z 131.971,A -85,B 0,C 180,E1 -20548.339,E2 -20548.339} C_VEL
LIN {X 0,Y 213.814,Z 132.18,A -85,B 0,C 180,E1 -20551.283,E2 -20551.283} C_VEL
LIN {X 0,Y 214.476,Z 134.256,A -85,B 0,C 180,E1 -20552.869,E2 -20552.869} C_VEL
LIN {X 0,Y 218.019,Z 139.185,A -85,B 0,C 180,E1 -20554.737,E2 -20554.737} C_VEL
LIN {X 0,Y 219.421,Z 140.887,A -85,B 0,C 180,E1 -20555.418,E2 -20555.418} C_VEL
LIN {X 0,Y 222.64,Z 145.415,A -85,B 0,C 180,E1 -20556.938,E2 -20556.938} C_VEL
LIN {X 0,Y 227.859,Z 153.249,A -85,B 0,C 180,E1 -20559.227,E2 -20559.227} C_VEL
LIN {X 0,Y 233.661,Z 162.283,A -85,B 0,C 180,E1 -20561.538,E2 -20561.538} C_VEL
LIN {X 0,Y 240.933,Z 174.941,A -85,B 0,C 180,E1 -20564.193,E2 -20564.193} C_VEL
LIN {X 0,Y 247.86,Z 188.732,A -85,B 0,C 180,E1 -20566.533,E2 -20566.533} C_VEL
LIN {X 0,Y 254.242,Z 203.426,A -85,B 0,C 180,E1 -20568.574,E2 -20568.574} C_VEL
LIN {X 0,Y 250.285,Z 273.844,A -85,B 0,C 180,E1 -20570.492,E2 -20570.492} C_VEL
LIN {X 0,Y 248.663,Z 287.458,A -85,B 0,C 180,E1 -20571.099,E2 -20571.099} C_VEL
LIN {X 0,Y 246.385,Z 300.364,A -85,B 0,C 180,E1 -20571.914,E2 -20571.914} C_VEL
LIN {X 0,Y 243.659,Z 312.742,A -85,B 0,C 180,E1 -20572.979,E2 -20572.979} C_VEL
LIN {X 0,Y 240.129,Z 325.688,A -85,B 0,C 180,E1 -20574.43,E2 -20574.43} C_VEL
LIN {X 0,Y 236.547,Z 337.276,A -85,B 0,C 180,E1 -20576.111,E2 -20576.111} C_VEL
LIN {X 0,Y 232.756,Z 348.189,A -85,B 0,C 180,E1 -20578.102,E2 -20578.102} C_VEL
LIN {X 0,Y 228.538,Z 358.846,A -85,B 0,C 180,E1 -20580.526,E2 -20580.526} C_VEL
LIN {X 0,Y 224.803,Z 367.658,A -85,B 0,C 180,E1 -20583.043,E2 -20583.043} C_VEL
LIN {X 0,Y 220.951,Z 376.12,A -85,B 0,C 180,E1 -20586.074,E2 -20586.074} C_VEL
LIN {X 0,Y 217.418,Z 383.748,A -85,B 0,C 180,E1 -20589.622,E2 -20589.622} C_VEL
LIN {X 0,Y 215.116,Z 389.087,A -85,B 0,C 180,E1 -20592.9,E2 -20592.9} C_VEL
LIN {X 0,Y 213.069,Z 393.597,A -85,B 0,C 180,E1 -20596.65,E2 -20596.65} C_VEL
LIN {X 0,Y 211.946,Z 396.676,A -85,B 0,C 180,E1 -20600.456,E2 -20600.456} C_VEL
LIN {X 0,Y 211.43,Z 398.402,A -85,B 0,C 180,E1 -20604.277,E2 -20604.277} C_VEL
LIN {X 0,Y 211.412,Z 398.803,A -85,B 0,C 180,E1 -20608.095,E2 -20608.095} C_VEL
LIN {X 0,Y 211.505,Z 398.506,A -85,B 0,C 180,E1 -20610,E2 -20610} C_VEL
LIN {X 0,Y 211.349,Z 396.888,A -85,B 0,C 180,E1 -20613.813,E2 -20613.813} C_VEL
LIN {X 0,Y 211.591,Z 393.884,A -85,B 0,C 180,E1 -20617.635,E2 -20617.635} C_VEL
LIN {X 0,Y 212.262,Z 389.401,A -85,B 0,C 180,E1 -20621.458,E2 -20621.458} C_VEL
LIN {X 0,Y 213.235,Z 384.948,A -85,B 0,C 180,E1 -20624.311,E2 -20624.311} C_VEL
LIN {X 0,Y 214.937,Z 378.502,A -85,B 0,C 180,E1 -20627.605,E2 -20627.605} C_VEL
LIN {X 0,Y 216.995,Z 370.465,A -85,B 0,C 180,E1 -20630.871,E2 -20630.871} C_VEL
LIN {X 0,Y 219.472,Z 362.063,A -85,B 0,C 180,E1 -20633.595,E2 -20633.595} C_VEL
LIN {X 0,Y 222.384,Z 351.935,A -85,B 0,C 180,E1 -20636.259,E2 -20636.259} C_VEL
LIN {X 0,Y 225.491,Z 340.615,A -85,B 0,C 180,E1 -20638.633,E2 -20638.633} C_VEL
LIN {X 0,Y 228.362,Z 328.762,A -85,B 0,C 180,E1 -20640.617,E2 -20640.617} C_VEL
LIN {X 0,Y 230.932,Z 317.009,A -85,B 0,C 180,E1 -20642.18,E2 -20642.18} C_VEL
LIN {X 0,Y 233.318,Z 304.439,A -85,B 0,C 180,E1 -20643.477,E2 -20643.477} C_VEL
LIN {X 0,Y 235.408,Z 290.396,A -85,B 0,C 180,E1 -20644.557,E2 -20644.557} C_VEL
LIN {X 0,Y 236.952,Z 275.608,A -85,B 0,C 180,E1 -20645.336,E2 -20645.336} C_VEL
LIN {X 0,Y 238.224,Z 252.983,A -85,B 0,C 180,E1 -20646.028,E2 -20646.028} C_VEL
LIN {X 0,Y 240.759,Z 194.375,A -85,B 0,C 180,E1 -20647.699,E2 -20647.699} C_VEL
LIN {X 0,Y 239.717,Z 187.269,A -85,B 0,C 180,E1 -20648.128,E2 -20648.128} C_VEL
LIN {X 0,Y 233.408,Z 171.301,A -85,B 0,C 180,E1 -20649.831,E2 -20649.831} C_VEL
LIN {X 0,Y 226.562,Z 156.592,A -85,B 0,C 180,E1 -20651.729,E2 -20651.729} C_VEL
LIN {X 0,Y 219.411,Z 143.488,A -85,B 0,C 180,E1 -20653.803,E2 -20653.803} C_VEL
LIN {X 0,Y 216.662,Z 138.883,A -85,B 0,C 180,E1 -20654.635,E2 -20654.635} C_VEL
LIN {X 0,Y 214.641,Z 134.997,A -85,B 0,C 180,E1 -20655.337,E2 -20655.337} C_VEL
LIN {X 0,Y 213.822,Z 131.971,A -85,B 0,C 180,E1 -20656.998,E2 -20656.998} C_VEL
LIN {X 0,Y 213.782,Z 131.954,A -85,B 0,C 180,E1 -20662.091,E2 -20662.091} C_VEL
LIN {X 0,Y 213.768,Z 131.975,A -85,B 0,C 180,E1 -20666.02,E2 -20666.02} C_VEL
LIN {X 0,Y 213.78,Z 131.973,A -85,B 0,C 180,E1 -20670.454,E2 -20670.454} C_VEL
LIN {X 0,Y 213.801,Z 131.971,A -85,B 0,C 180,E1 -20674.702,E2 -20674.702} C_VEL
LIN {X 0,Y 213.813,Z 131.977,A -85,B 0,C 180,E1 -20678.804,E2 -20678.804} C_VEL
LIN {X 0,Y 213.943,Z 131.953,A -85,B 0,C 180,E1 -20682.804,E2 -20682.804} C_VEL
LIN {X 0,Y 213.954,Z 131.945,A -85,B 0,C 180,E1 -20686.707,E2 -20686.707} C_VEL
LIN {X 0,Y 214.163,Z 131.934,A -85,B 0,C 180,E1 -20690.556,E2 -20690.556} C_VEL
LIN {X 0,Y 214.222,Z 131.919,A -85,B 0,C 180,E1 -20692.46,E2 -20692.46} C_VEL
LIN {X 0,Y 214.445,Z 131.899,A -85,B 0,C 180,E1 -20698.122,E2 -20698.122} C_VEL
LIN {X 0,Y 214.549,Z 131.874,A -85,B 0,C 180,E1 -20700,E2 -20700} C_VEL
LIN {X 0,Y 214.443,Z 131.875,A -85,B 0,C 180,E1 -20701.878,E2 -20701.878} C_VEL
LIN {X 0,Y 214.188,Z 131.925,A -85,B 0,C 180,E1 -20707.542,E2 -20707.542} C_VEL
LIN {X 0,Y 213.999,Z 131.939,A -85,B 0,C 180,E1 -20711.365,E2 -20711.365} C_VEL
LIN {X 0,Y 213.934,Z 131.958,A -85,B 0,C 180,E1 -20715.237,E2 -20715.237} C_VEL
LIN {X 0,Y 213.876,Z 131.957,A -85,B 0,C 180,E1 -20719.184,E2 -20719.184} C_VEL
LIN {X 0,Y 213.856,Z 131.963,A -85,B 0,C 180,E1 -20723.226,E2 -20723.226} C_VEL
LIN {X 0,Y 213.829,Z 131.972,A -85,B 0,C 180,E1 -20727.45,E2 -20727.45} C_VEL
LIN {X 0,Y 213.768,Z 131.968,A -85,B 0,C 180,E1 -20731.738,E2 -20731.738} C_VEL
LIN {X 0,Y 213.744,Z 131.976,A -85,B 0,C 180,E1 -20736.289,E2 -20736.289} C_VEL
LIN {X 0,Y 213.713,Z 131.98,A -85,B 0,C 180,E1 -20741.126,E2 -20741.126} C_VEL
LIN {X 0,Y 213.708,Z 131.99,A -85,B 0,C 180,E1 -20743.679,E2 -20743.679} C_VEL
LIN {X 0,Y 213.708,Z 131.981,A -85,B 0,C 180,E1 -20746.344,E2 -20746.344} C_VEL
LIN {X 0,Y 213.779,Z 131.953,A -85,B 0,C 180,E1 -20750.718,E2 -20750.718} C_VEL
LIN {X 0,Y 214.71,Z 134.745,A -85,B 0,C 180,E1 -20751.091,E2 -20751.091} C_VEL
LIN {X 0,Y 216.755,Z 137.304,A -85,B 0,C 180,E1 -20751.694,E2 -20751.694} C_VEL
LIN {X 0,Y 219.08,Z 140.776,A -85,B 0,C 180,E1 -20752.382,E2 -20752.382} C_VEL
LIN {X 0,Y 228.473,Z 156.028,A -85,B 0,C 180,E1 -20755.009,E2 -20755.009} C_VEL
LIN {X 0,Y 232.116,Z 163.007,A -85,B 0,C 180,E1 -20755.987,E2 -20755.987} C_VEL
LIN {X 0,Y 238.891,Z 178.487,A -85,B 0,C 180,E1 -20757.789,E2 -20757.789} C_VEL
LIN {X 0,Y 241.177,Z 184.381,A -85,B 0,C 180,E1 -20758.389,E2 -20758.389} C_VEL
LIN {X 0,Y 237.469,Z 264.876,A -85,B 0,C 180,E1 -20760.709,E2 -20760.709} C_VEL
LIN {X 0,Y 236.28,Z 278.488,A -85,B 0,C 180,E1 -20761.4,E2 -20761.4} C_VEL
LIN {X 0,Y 234.612,Z 291.38,A -85,B 0,C 180,E1 -20762.334,E2 -20762.334} C_VEL
LIN {X 0,Y 232.545,Z 303.755,A -85,B 0,C 180,E1 -20763.527,E2 -20763.527} C_VEL
LIN {X 0,Y 229.853,Z 316.688,A -85,B 0,C 180,E1 -20765.139,E2 -20765.139} C_VEL
LIN {X 0,Y 227.18,Z 328.392,A -85,B 0,C 180,E1 -20767.011,E2 -20767.011} C_VEL
LIN {X 0,Y 224.114,Z 340.079,A -85,B 0,C 180,E1 -20769.342,E2 -20769.342} C_VEL
LIN {X 0,Y 221.121,Z 350.527,A -85,B 0,C 180,E1 -20771.948,E2 -20771.948} C_VEL
LIN {X 0,Y 218.622,Z 359.279,A -85,B 0,C 180,E1 -20774.669,E2 -20774.669} C_VEL
LIN {X 0,Y 216.278,Z 367.42,A -85,B 0,C 180,E1 -20777.807,E2 -20777.807} C_VEL
LIN {X 0,Y 214.541,Z 373.191,A -85,B 0,C 180,E1 -20780.573,E2 -20780.573} C_VEL
LIN {X 0,Y 212.863,Z 379.368,A -85,B 0,C 180,E1 -20784.316,E2 -20784.316} C_VEL
LIN {X 0,Y 211.959,Z 383.904,A -85,B 0,C 180,E1 -20788.1,E2 -20788.1} C_VEL
LIN {X 0,Y 211.505,Z 386.99,A -85,B 0,C 180,E1 -20791.905,E2 -20791.905} C_VEL
LIN {X 0,Y 211.421,Z 388.203,A -85,B 0,C 180,E1 -20794.242,E2 -20794.242} C_VEL
LIN {X 0,Y 211.358,Z 389.098,A -85,B 0,C 180,E1 -20797.644,E2 -20797.644} C_VEL
LIN {X 0,Y 211.54,Z 388.853,A -85,B 0,C 180,E1 -20801.499,E2 -20801.499} C_VEL
LIN {X 0,Y 212.438,Z 387.266,A -85,B 0,C 180,E1 -20805.347,E2 -20805.347} C_VEL
LIN {X 0,Y 213.863,Z 384.297,A -85,B 0,C 180,E1 -20809.185,E2 -20809.185} C_VEL
LIN {X 0,Y 216.056,Z 379.855,A -85,B 0,C 180,E1 -20812.976,E2 -20812.976} C_VEL
LIN {X 0,Y 218.347,Z 375.157,A -85,B 0,C 180,E1 -20815.92,E2 -20815.92} C_VEL
LIN {X 0,Y 221.782,Z 367.958,A -85,B 0,C 180,E1 -20819.418,E2 -20819.418} C_VEL
LIN {X 0,Y 225.014,Z 360.938,A -85,B 0,C 180,E1 -20822.071,E2 -20822.071} C_VEL
LIN {X 0,Y 228.581,Z 352.493,A -85,B 0,C 180,E1 -20824.667,E2 -20824.667} C_VEL
LIN {X 0,Y 232.649,Z 342.285,A -85,B 0,C 180,E1 -20827.17,E2 -20827.17} C_VEL
LIN {X 0,Y 236.332,Z 332.456,A -85,B 0,C 180,E1 -20829.074,E2 -20829.074} C_VEL
LIN {X 0,Y 239.977,Z 320.755,A -85,B 0,C 180,E1 -20830.941,E2 -20830.941} C_VEL
LIN {X 0,Y 243.478,Z 308.519,A -85,B 0,C 180,E1 -20832.433,E2 -20832.433} C_VEL
LIN {X 0,Y 246.243,Z 296.012,A -85,B 0,C 180,E1 -20833.657,E2 -20833.657} C_VEL
LIN {X 0,Y 248.633,Z 282.028,A -85,B 0,C 180,E1 -20834.679,E2 -20834.679} C_VEL
LIN {X 0,Y 250.459,Z 267.384,A -85,B 0,C 180,E1 -20835.4,E2 -20835.4} C_VEL
LIN {X 0,Y 251.854,Z 246,A -85,B 0,C 180,E1 -20836.035,E2 -20836.035} C_VEL
LIN {X 0,Y 254.608,Z 197.299,A -85,B 0,C 180,E1 -20837.311,E2 -20837.311} C_VEL
LIN {X 0,Y 247.858,Z 183.056,A -85,B 0,C 180,E1 -20839.428,E2 -20839.428} C_VEL
LIN {X 0,Y 241.47,Z 171.063,A -85,B 0,C 180,E1 -20841.562,E2 -20841.562} C_VEL
LIN {X 0,Y 236.592,Z 163.008,A -85,B 0,C 180,E1 -20843.286,E2 -20843.286} C_VEL
LIN {X 0,Y 231.303,Z 155.505,A -85,B 0,C 180,E1 -20845.255,E2 -20845.255} C_VEL
LIN {X 0,Y 228.324,Z 151.415,A -85,B 0,C 180,E1 -20846.439,E2 -20846.439} C_VEL
LIN {X 0,Y 225.241,Z 147.248,A -85,B 0,C 180,E1 -20847.731,E2 -20847.731} C_VEL
LIN {X 0,Y 222.551,Z 143.78,A -85,B 0,C 180,E1 -20848.915,E2 -20848.915} C_VEL
LIN {X 0,Y 221.647,Z 142.589,A -85,B 0,C 180,E1 -20849.329,E2 -20849.329} C_VEL
LIN {X 0,Y 219.171,Z 139.939,A -85,B 0,C 180,E1 -20850.469,E2 -20850.469} C_VEL
LIN {X 0,Y 217.806,Z 137.511,A -85,B 0,C 180,E1 -20851.184,E2 -20851.184} C_VEL
LIN {X 0,Y 215.439,Z 135.712,A -85,B 0,C 180,E1 -20852.328,E2 -20852.328} C_VEL
LIN {X 0,Y 214.136,Z 133.284,A -85,B 0,C 180,E1 -20853.08,E2 -20853.08} C_VEL
LIN {X 0,Y 213.835,Z 131.963,A -85,B 0,C 180,E1 -20853.397,E2 -20853.397} C_VEL
LIN {X 0,Y 213.812,Z 131.966,A -85,B 0,C 180,E1 -20856.979,E2 -20856.979} C_VEL
LIN {X 0,Y 213.923,Z 131.952,A -85,B 0,C 180,E1 -20862.802,E2 -20862.802} C_VEL
LIN {X 0,Y 213.945,Z 131.945,A -85,B 0,C 180,E1 -20866.706,E2 -20866.706} C_VEL
LIN {X 0,Y 214.135,Z 131.921,A -85,B 0,C 180,E1 -20870.555,E2 -20870.555} C_VEL
LIN {X 0,Y 214.087,Z 131.939,A -85,B 0,C 180,E1 -20874.348,E2 -20874.348} C_VEL
LIN {X 0,Y 214.443,Z 131.895,A -85,B 0,C 180,E1 -20878.122,E2 -20878.122} C_VEL
LIN {X 0,Y 214.547,Z 131.874,A -85,B 0,C 180,E1 -20880,E2 -20880} C_VEL
LIN {X 0,Y 214.443,Z 131.882,A -85,B 0,C 180,E1 -20881.878,E2 -20881.878} C_VEL
LIN {X 0,Y 214.187,Z 131.918,A -85,B 0,C 180,E1 -20887.542,E2 -20887.542} C_VEL
LIN {X 0,Y 214.001,Z 131.937,A -85,B 0,C 180,E1 -20891.364,E2 -20891.364} C_VEL
LIN {X 0,Y 213.935,Z 131.948,A -85,B 0,C 180,E1 -20895.237,E2 -20895.237} C_VEL
LIN {X 0,Y 213.841,Z 131.966,A -85,B 0,C 180,E1 -20899.187,E2 -20899.187} C_VEL
LIN {X 0,Y 213.849,Z 131.968,A -85,B 0,C 180,E1 -20903.227,E2 -20903.227} C_VEL
LIN {X 0,Y 213.766,Z 131.971,A -85,B 0,C 180,E1 -20908.339,E2 -20908.339} C_VEL
LIN {X 0,Y 213.75,Z 132.514,A -85,B 0,C 180,E1 -20909.367,E2 -20909.367} C_VEL
LIN {X 0,Y 213.88,Z 134.856,A -85,B 0,C 180,E1 -20910.808,E2 -20910.808} C_VEL
LIN {X 0,Y 214.287,Z 138.301,A -85,B 0,C 180,E1 -20912.101,E2 -20912.101} C_VEL
LIN {X 0,Y 215.52,Z 143.783,A -85,B 0,C 180,E1 -20913.721,E2 -20913.721} C_VEL
LIN {X 0,Y 217.214,Z 147.706,A -85,B 0,C 180,E1 -20914.904,E2 -20914.904} C_VEL
LIN {X 0,Y 217.977,Z 148.868,A -85,B 0,C 180,E1 -20915.304,E2 -20915.304} C_VEL
LIN {X 0,Y 220.785,Z 152.704,A -85,B 0,C 180,E1 -20916.644,E2 -20916.644} C_VEL
LIN {X 0,Y 224.805,Z 158.948,A -85,B 0,C 180,E1 -20918.471,E2 -20918.471} C_VEL
LIN {X 0,Y 230.315,Z 167.77,A -85,B 0,C 180,E1 -20920.767,E2 -20920.767} C_VEL
LIN {X 0,Y 236.531,Z 178.769,A -85,B 0,C 180,E1 -20923.153,E2 -20923.153} C_VEL
LIN {X 0,Y 243.351,Z 192.481,A -85,B 0,C 180,E1 -20925.58,E2 -20925.58} C_VEL
LIN {X 0,Y 249.111,Z 205.897,A -85,B 0,C 180,E1 -20927.522,E2 -20927.522} C_VEL
LIN {X 0,Y 245.115,Z 273.148,A -85,B 0,C 180,E1 -20929.353,E2 -20929.353} C_VEL
LIN {X 0,Y 243.454,Z 286.935,A -85,B 0,C 180,E1 -20929.968,E2 -20929.968} C_VEL
LIN {X 0,Y 241.118,Z 299.931,A -85,B 0,C 180,E1 -20930.792,E2 -20930.792} C_VEL
LIN {X 0,Y 238.483,Z 311.464,A -85,B 0,C 180,E1 -20931.767,E2 -20931.767} C_VEL
LIN {X 0,Y 234.819,Z 324.647,A -85,B 0,C 180,E1 -20933.231,E2 -20933.231} C_VEL
LIN {X 0,Y 231.048,Z 336.548,A -85,B 0,C 180,E1 -20934.961,E2 -20934.961} C_VEL
LIN {X 0,Y 227.508,Z 346.453,A -85,B 0,C 180,E1 -20936.748,E2 -20936.748} C_VEL
LIN {X 0,Y 223.102,Z 357.367,A -85,B 0,C 180,E1 -20939.21,E2 -20939.21} C_VEL
LIN {X 0,Y 219.06,Z 366.4,A -85,B 0,C 180,E1 -20941.756,E2 -20941.756} C_VEL
LIN {X 0,Y 215.005,Z 375.053,A -85,B 0,C 180,E1 -20944.853,E2 -20944.853} C_VEL
LIN {X 0,Y 212.013,Z 381.153,A -85,B 0,C 180,E1 -20947.591,E2 -20947.591} C_VEL
LIN {X 0,Y 209.65,Z 386.222,A -85,B 0,C 180,E1 -20950.413,E2 -20950.413} C_VEL
LIN {X 0,Y 207.129,Z 391.466,A -85,B 0,C 180,E1 -20954.25,E2 -20954.25} C_VEL
LIN {X 0,Y 205.436,Z 395.214,A -85,B 0,C 180,E1 -20958.155,E2 -20958.155} C_VEL
LIN {X 0,Y 204.561,Z 397.579,A -85,B 0,C 180,E1 -20962.101,E2 -20962.101} C_VEL
LIN {X 0,Y 204.296,Z 398.613,A -85,B 0,C 180,E1 -20966.054,E2 -20966.054} C_VEL
LIN {X 0,Y 204.406,Z 398.32,A -85,B 0,C 180,E1 -20970,E2 -20970} C_VEL
LIN {X 0,Y 204.259,Z 396.672,A -85,B 0,C 180,E1 -20973.946,E2 -20973.946} C_VEL
LIN {X 0,Y 204.532,Z 393.636,A -85,B 0,C 180,E1 -20977.9,E2 -20977.9} C_VEL
LIN {X 0,Y 205.252,Z 389.119,A -85,B 0,C 180,E1 -20981.855,E2 -20981.855} C_VEL
LIN {X 0,Y 206.321,Z 384.631,A -85,B 0,C 180,E1 -20984.801,E2 -20984.801} C_VEL
LIN {X 0,Y 207.821,Z 379.163,A -85,B 0,C 180,E1 -20987.719,E2 -20987.719} C_VEL
LIN {X 0,Y 209.941,Z 371.31,A -85,B 0,C 180,E1 -20991.092,E2 -20991.092} C_VEL
LIN {X 0,Y 212.454,Z 363.114,A -85,B 0,C 180,E1 -20993.905,E2 -20993.905} C_VEL
LIN {X 0,Y 215.413,Z 353.226,A -85,B 0,C 180,E1 -20996.654,E2 -20996.654} C_VEL
LIN {X 0,Y 218.665,Z 342.243,A -85,B 0,C 180,E1 -20999.086,E2 -20999.086} C_VEL
LIN {X 0,Y 221.715,Z 330.237,A -85,B 0,C 180,E1 -21001.227,E2 -21001.227} C_VEL
LIN {X 0,Y 224.554,Z 317.94,A -85,B 0,C 180,E1 -21002.942,E2 -21002.942} C_VEL
LIN {X 0,Y 227.215,Z 304.552,A -85,B 0,C 180,E1 -21004.366,E2 -21004.366} C_VEL
LIN {X 0,Y 229.361,Z 290.6,A -85,B 0,C 180,E1 -21005.469,E2 -21005.469} C_VEL
LIN {X 0,Y 230.972,Z 275.998,A -85,B 0,C 180,E1 -21006.259,E2 -21006.259} C_VEL
LIN {X 0,Y 232.184,Z 255.484,A -85,B 0,C 180,E1 -21006.916,E2 -21006.916} C_VEL
LIN {X 0,Y 234.926,Z 195.259,A -85,B 0,C 180,E1 -21008.662,E2 -21008.662} C_VEL
LIN {X 0,Y 234.042,Z 189.573,A -85,B 0,C 180,E1 -21009.03,E2 -21009.03} C_VEL
LIN {X 0,Y 228.028,Z 174.403,A -85,B 0,C 180,E1 -21010.733,E2 -21010.733} C_VEL
LIN {X 0,Y 221.829,Z 160.83,A -85,B 0,C 180,E1 -21012.545,E2 -21012.545} C_VEL
LIN {X 0,Y 215.041,Z 148.134,A -85,B 0,C 180,E1 -21014.614,E2 -21014.614} C_VEL
LIN {X 0,Y 209.731,Z 139.115,A -85,B 0,C 180,E1 -21016.334,E2 -21016.334} C_VEL
LIN {X 0,Y 207.727,Z 135.752,A -85,B 0,C 180,E1 -21017.018,E2 -21017.018} C_VEL
LIN {X 0,Y 207.321,Z 134.817,A -85,B 0,C 180,E1 -21017.2,E2 -21017.2} C_VEL
LIN {X 0,Y 206.746,Z 132.857,A -85,B 0,C 180,E1 -21018.404,E2 -21018.404} C_VEL
LIN {X 0,Y 206.724,Z 132.833,A -85,B 0,C 180,E1 -21022.27,E2 -21022.27} C_VEL
LIN {X 0,Y 206.708,Z 132.853,A -85,B 0,C 180,E1 -21027.044,E2 -21027.044} C_VEL
LIN {X 0,Y 206.766,Z 132.85,A -85,B 0,C 180,E1 -21032.096,E2 -21032.096} C_VEL
LIN {X 0,Y 206.785,Z 132.842,A -85,B 0,C 180,E1 -21036.584,E2 -21036.584} C_VEL
LIN {X 0,Y 206.873,Z 132.83,A -85,B 0,C 180,E1 -21042.197,E2 -21042.197} C_VEL
LIN {X 0,Y 206.896,Z 132.828,A -85,B 0,C 180,E1 -21046.245,E2 -21046.245} C_VEL
LIN {X 0,Y 207.102,Z 132.811,A -85,B 0,C 180,E1 -21050.231,E2 -21050.231} C_VEL
LIN {X 0,Y 207.068,Z 132.799,A -85,B 0,C 180,E1 -21054.156,E2 -21054.156} C_VEL
LIN {X 0,Y 207.381,Z 132.779,A -85,B 0,C 180,E1 -21058.058,E2 -21058.058} C_VEL
LIN {X 0,Y 207.514,Z 132.75,A -85,B 0,C 180,E1 -21060,E2 -21060} C_VEL
LIN {X 0,Y 207.379,Z 132.754,A -85,B 0,C 180,E1 -21061.942,E2 -21061.942} C_VEL
LIN {X 0,Y 207.132,Z 132.8,A -85,B 0,C 180,E1 -21067.801,E2 -21067.801} C_VEL
LIN {X 0,Y 206.925,Z 132.822,A -85,B 0,C 180,E1 -21071.759,E2 -21071.759} C_VEL
LIN {X 0,Y 206.868,Z 132.833,A -85,B 0,C 180,E1 -21075.771,E2 -21075.771} C_VEL
LIN {X 0,Y 206.813,Z 132.841,A -85,B 0,C 180,E1 -21079.867,E2 -21079.867} C_VEL
LIN {X 0,Y 206.768,Z 132.838,A -85,B 0,C 180,E1 -21084.072,E2 -21084.072} C_VEL
LIN {X 0,Y 206.744,Z 132.857,A -85,B 0,C 180,E1 -21088.419,E2 -21088.419} C_VEL
LIN {X 0,Y 206.699,Z 132.855,A -85,B 0,C 180,E1 -21092.958,E2 -21092.958} C_VEL
LIN {X 0,Y 206.68,Z 132.855,A -85,B 0,C 180,E1 -21097.74,E2 -21097.74} C_VEL
LIN {X 0,Y 206.643,Z 132.859,A -85,B 0,C 180,E1 -21101.564,E2 -21101.564} C_VEL
LIN {X 0,Y 206.635,Z 132.862,A -85,B 0,C 180,E1 -21105.582,E2 -21105.582} C_VEL
LIN {X 0,Y 206.682,Z 132.956,A -85,B 0,C 180,E1 -21108.945,E2 -21108.945} C_VEL
LIN {X 0,Y 207.664,Z 135.675,A -85,B 0,C 180,E1 -21109.339,E2 -21109.339} C_VEL
LIN {X 0,Y 209.828,Z 138.272,A -85,B 0,C 180,E1 -21110.028,E2 -21110.028} C_VEL
LIN {X 0,Y 212.108,Z 141.69,A -85,B 0,C 180,E1 -21110.762,E2 -21110.762} C_VEL
LIN {X 0,Y 219.77,Z 153.594,A -85,B 0,C 180,E1 -21113.08,E2 -21113.08} C_VEL
LIN {X 0,Y 226.079,Z 164.666,A -85,B 0,C 180,E1 -21114.87,E2 -21114.87} C_VEL
LIN {X 0,Y 232.786,Z 179.722,A -85,B 0,C 180,E1 -21116.748,E2 -21116.748} C_VEL
LIN {X 0,Y 235.221,Z 186.119,A -85,B 0,C 180,E1 -21117.427,E2 -21117.427} C_VEL
LIN {X 0,Y 233.863,Z 218.638,A -85,B 0,C 180,E1 -21118.391,E2 -21118.391} C_VEL
LIN {X 0,Y 231.553,Z 264.909,A -85,B 0,C 180,E1 -21119.759,E2 -21119.759} C_VEL
LIN {X 0,Y 230.316,Z 278.563,A -85,B 0,C 180,E1 -21120.462,E2 -21120.462} C_VEL
LIN {X 0,Y 228.559,Z 291.483,A -85,B 0,C 180,E1 -21121.411,E2 -21121.411} C_VEL
LIN {X 0,Y 226.25,Z 304.746,A -85,B 0,C 180,E1 -21122.731,E2 -21122.731} C_VEL
LIN {X 0,Y 223.476,Z 317.518,A -85,B 0,C 180,E1 -21124.379,E2 -21124.379} C_VEL
LIN {X 0,Y 220.701,Z 329.105,A -85,B 0,C 180,E1 -21126.295,E2 -21126.295} C_VEL
LIN {X 0,Y 218.123,Z 338.757,A -85,B 0,C 180,E1 -21128.252,E2 -21128.252} C_VEL
LIN {X 0,Y 214.902,Z 349.455,A -85,B 0,C 180,E1 -21130.912,E2 -21130.912} C_VEL
LIN {X 0,Y 212.297,Z 358.279,A -85,B 0,C 180,E1 -21133.658,E2 -21133.658} C_VEL
LIN {X 0,Y 209.739,Z 366.735,A -85,B 0,C 180,E1 -21136.928,E2 -21136.928} C_VEL
LIN {X 0,Y 207.557,Z 373.566,A -85,B 0,C 180,E1 -21140.253,E2 -21140.253} C_VEL
LIN {X 0,Y 206.229,Z 378.283,A -85,B 0,C 180,E1 -21143.15,E2 -21143.15} C_VEL
LIN {X 0,Y 205.09,Z 383.175,A -85,B 0,C 180,E1 -21147.054,E2 -21147.054} C_VEL
LIN {X 0,Y 204.601,Z 385.868,A -85,B 0,C 180,E1 -21150,E2 -21150} C_VEL
LIN {X 0,Y 204.328,Z 388.282,A -85,B 0,C 180,E1 -21154.067,E2 -21154.067} C_VEL
LIN {X 0,Y 204.261,Z 389.271,A -85,B 0,C 180,E1 -21157.911,E2 -21157.911} C_VEL
LIN {X 0,Y 204.497,Z 388.989,A -85,B 0,C 180,E1 -21161.9,E2 -21161.9} C_VEL
LIN {X 0,Y 205.506,Z 387.363,A -85,B 0,C 180,E1 -21165.878,E2 -21165.878} C_VEL
LIN {X 0,Y 207.035,Z 384.356,A -85,B 0,C 180,E1 -21169.844,E2 -21169.844} C_VEL
LIN {X 0,Y 209.407,Z 379.871,A -85,B 0,C 180,E1 -21173.75,E2 -21173.75} C_VEL
LIN {X 0,Y 211.731,Z 375.347,A -85,B 0,C 180,E1 -21176.65,E2 -21176.65} C_VEL
LIN {X 0,Y 214.978,Z 368.896,A -85,B 0,C 180,E1 -21179.904,E2 -21179.904} C_VEL
LIN {X 0,Y 218.903,Z 360.807,A -85,B 0,C 180,E1 -21183.079,E2 -21183.079} C_VEL
LIN {X 0,Y 222.662,Z 352.301,A -85,B 0,C 180,E1 -21185.727,E2 -21185.727} C_VEL
LIN {X 0,Y 226.936,Z 341.99,A -85,B 0,C 180,E1 -21188.271,E2 -21188.271} C_VEL
LIN {X 0,Y 231.099,Z 331.153,A -85,B 0,C 180,E1 -21190.364,E2 -21190.364} C_VEL
LIN {X 0,Y 234.576,Z 320.239,A -85,B 0,C 180,E1 -21192.095,E2 -21192.095} C_VEL
LIN {X 0,Y 238.207,Z 307.838,A -85,B 0,C 180,E1 -21193.603,E2 -21193.603} C_VEL
LIN {X 0,Y 241.099,Z 295.1,A -85,B 0,C 180,E1 -21194.835,E2 -21194.835} C_VEL
LIN {X 0,Y 243.582,Z 280.743,A -85,B 0,C 180,E1 -21195.866,E2 -21195.866} C_VEL
LIN {X 0,Y 245.278,Z 267.234,A -85,B 0,C 180,E1 -21196.521,E2 -21196.521} C_VEL
LIN {X 0,Y 246.812,Z 244.585,A -85,B 0,C 180,E1 -21197.187,E2 -21197.187} C_VEL
LIN {X 0,Y 249.383,Z 199.721,A -85,B 0,C 180,E1 -21198.391,E2 -21198.391} C_VEL
LIN {X 0,Y 242.922,Z 185.89,A -85,B 0,C 180,E1 -21200.538,E2 -21200.538} C_VEL
LIN {X 0,Y 236.75,Z 174.369,A -85,B 0,C 180,E1 -21202.715,E2 -21202.715} C_VEL
LIN {X 0,Y 233.025,Z 168.165,A -85,B 0,C 180,E1 -21204.101,E2 -21204.101} C_VEL
LIN {X 0,Y 227.207,Z 159.836,A -85,B 0,C 180,E1 -21206.38,E2 -21206.38} C_VEL
LIN {X 0,Y 224.936,Z 156.707,A -85,B 0,C 180,E1 -21207.331,E2 -21207.331} C_VEL
LIN {X 0,Y 222.083,Z 152.828,A -85,B 0,C 180,E1 -21208.584,E2 -21208.584} C_VEL
LIN {X 0,Y 218.909,Z 148.642,A -85,B 0,C 180,E1 -21210.059,E2 -21210.059} C_VEL
LIN {X 0,Y 216.223,Z 145.431,A -85,B 0,C 180,E1 -21211.371,E2 -21211.371} C_VEL
LIN {X 0,Y 215.071,Z 143.713,A -85,B 0,C 180,E1 -21211.981,E2 -21211.981} C_VEL
LIN {X 0,Y 212.675,Z 141.378,A -85,B 0,C 180,E1 -21213.226,E2 -21213.226} C_VEL
LIN {X 0,Y 211.207,Z 138.57,A -85,B 0,C 180,E1 -21214.123,E2 -21214.123} C_VEL
LIN {X 0,Y 208.531,Z 136.775,A -85,B 0,C 180,E1 -21215.615,E2 -21215.615} C_VEL
LIN {X 0,Y 207.157,Z 134.492,A -85,B 0,C 180,E1 -21216.531,E2 -21216.531} C_VEL
LIN {X 0,Y 206.765,Z 132.844,A -85,B 0,C 180,E1 -21216.894,E2 -21216.894} C_VEL
LIN {X 0,Y 206.87,Z 132.828,A -85,B 0,C 180,E1 -21222.196,E2 -21222.196} C_VEL
LIN {X 0,Y 206.886,Z 132.824,A -85,B 0,C 180,E1 -21226.243,E2 -21226.243} C_VEL
LIN {X 0,Y 207.08,Z 132.802,A -85,B 0,C 180,E1 -21230.23,E2 -21230.23} C_VEL
LIN {X 0,Y 207.049,Z 132.817,A -85,B 0,C 180,E1 -21234.155,E2 -21234.155} C_VEL
LIN {X 0,Y 207.379,Z 132.774,A -85,B 0,C 180,E1 -21238.058,E2 -21238.058} C_VEL
LIN {X 0,Y 207.512,Z 132.75,A -85,B 0,C 180,E1 -21240,E2 -21240} C_VEL
LIN {X 0,Y 207.379,Z 132.762,A -85,B 0,C 180,E1 -21241.942,E2 -21241.942} C_VEL
LIN {X 0,Y 207.131,Z 132.799,A -85,B 0,C 180,E1 -21247.8,E2 -21247.8} C_VEL
LIN {X 0,Y 206.926,Z 132.818,A -85,B 0,C 180,E1 -21251.758,E2 -21251.758} C_VEL
LIN {X 0,Y 206.868,Z 132.825,A -85,B 0,C 180,E1 -21255.77,E2 -21255.77} C_VEL
LIN {X 0,Y 206.785,Z 132.838,A -85,B 0,C 180,E1 -21259.869,E2 -21259.869} C_VEL
LIN {X 0,Y 206.765,Z 132.842,A -85,B 0,C 180,E1 -21264.072,E2 -21264.072} C_VEL
LIN {X 0,Y 206.758,Z 133.038,A -85,B 0,C 180,E1 -21268.416,E2 -21268.416} C_VEL
LIN {X 0,Y 206.92,Z 133.859,A -85,B 0,C 180,E1 -21269.016,E2 -21269.016} C_VEL
LIN {X 0,Y 208.057,Z 136.153,A -85,B 0,C 180,E1 -21269.814,E2 -21269.814} C_VEL
LIN {X 0,Y 211.986,Z 140.347,A -85,B 0,C 180,E1 -21272.106,E2 -21272.106} C_VEL
LIN {X 0,Y 215.702,Z 145.499,A -85,B 0,C 180,E1 -21274.136,E2 -21274.136} C_VEL
LIN {X 0,Y 217.036,Z 147.418,A -85,B 0,C 180,E1 -21274.825,E2 -21274.825} C_VEL
LIN {X 0,Y 217.977,Z 148.868,A -85,B 0,C 180,E1 -21275.304,E2 -21275.304} C_VEL
LIN {X 0,Y 220.05,Z 152.631,A -85,B 0,C 180,E1 -21276.355,E2 -21276.355} C_VEL
LIN {X 0,Y 221.692,Z 157.187,A -85,B 0,C 180,E1 -21277.242,E2 -21277.242} C_VEL
LIN {X 0,Y 225.67,Z 170.276,A -85,B 0,C 180,E1 -21279.37,E2 -21279.37} C_VEL
LIN {X 0,Y 227.008,Z 173.204,A -85,B 0,C 180,E1 -21279.97,E2 -21279.97} C_VEL
LIN {X 0,Y 233.442,Z 184.95,A -85,B 0,C 180,E1 -21282.549,E2 -21282.549} C_VEL
LIN {X 0,Y 239.856,Z 198.267,A -85,B 0,C 180,E1 -21284.93,E2 -21284.93} C_VEL
LIN {X 0,Y 244.049,Z 208.294,A -85,B 0,C 180,E1 -21286.419,E2 -21286.419} C_VEL
LIN {X 0,Y 239.938,Z 273.607,A -85,B 0,C 180,E1 -21288.212,E2 -21288.212} C_VEL
LIN {X 0,Y 238.216,Z 287.188,A -85,B 0,C 180,E1 -21288.831,E2 -21288.831} C_VEL
LIN {X 0,Y 235.693,Z 300.637,A -85,B 0,C 180,E1 -21289.707,E2 -21289.707} C_VEL
LIN {X 0,Y 232.977,Z 312.009,A -85,B 0,C 180,E1 -21290.692,E2 -21290.692} C_VEL
LIN {X 0,Y 229.196,Z 325.032,A -85,B 0,C 180,E1 -21292.173,E2 -21292.173} C_VEL
LIN {X 0,Y 225.248,Z 336.951,A -85,B 0,C 180,E1 -21293.947,E2 -21293.947} C_VEL
LIN {X 0,Y 221.605,Z 346.674,A -85,B 0,C 180,E1 -21295.745,E2 -21295.745} C_VEL
LIN {X 0,Y 217.022,Z 357.514,A -85,B 0,C 180,E1 -21298.248,E2 -21298.248} C_VEL
LIN {X 0,Y 212.817,Z 366.494,A -85,B 0,C 180,E1 -21300.85,E2 -21300.85} C_VEL
LIN {X 0,Y 208.578,Z 375.102,A -85,B 0,C 180,E1 -21304.021,E2 -21304.021} C_VEL
LIN {X 0,Y 205.424,Z 381.161,A -85,B 0,C 180,E1 -21306.831,E2 -21306.831} C_VEL
LIN {X 0,Y 202.913,Z 386.198,A -85,B 0,C 180,E1 -21309.735,E2 -21309.735} C_VEL
LIN {X 0,Y 200.266,Z 391.403,A -85,B 0,C 180,E1 -21313.695,E2 -21313.695} C_VEL
LIN {X 0,Y 198.461,Z 395.12,A -85,B 0,C 180,E1 -21317.732,E2 -21317.732} C_VEL
LIN {X 0,Y 197.499,Z 397.454,A -85,B 0,C 180,E1 -21321.816,E2 -21321.816} C_VEL
LIN {X 0,Y 197.205,Z 398.457,A -85,B 0,C 180,E1 -21325.912,E2 -21325.912} C_VEL
LIN {X 0,Y 197.309,Z 398.135,A -85,B 0,C 180,E1 -21330,E2 -21330} C_VEL
LIN {X 0,Y 197.172,Z 396.456,A -85,B 0,C 180,E1 -21334.088,E2 -21334.088} C_VEL
LIN {X 0,Y 197.47,Z 393.388,A -85,B 0,C 180,E1 -21338.184,E2 -21338.184} C_VEL
LIN {X 0,Y 198.26,Z 388.834,A -85,B 0,C 180,E1 -21342.28,E2 -21342.28} C_VEL
LIN {X 0,Y 199.427,Z 384.313,A -85,B 0,C 180,E1 -21345.325,E2 -21345.325} C_VEL
LIN {X 0,Y 201.465,Z 377.109,A -85,B 0,C 180,E1 -21349.175,E2 -21349.175} C_VEL
LIN {X 0,Y 203.686,Z 369.666,A -85,B 0,C 180,E1 -21352.305,E2 -21352.305} C_VEL
LIN {X 0,Y 206.394,Z 361.164,A -85,B 0,C 180,E1 -21355.191,E2 -21355.191} C_VEL
LIN {X 0,Y 209.667,Z 350.907,A -85,B 0,C 180,E1 -21357.987,E2 -21357.987} C_VEL
LIN {X 0,Y 213.011,Z 339.4,A -85,B 0,C 180,E1 -21360.479,E2 -21360.479} C_VEL
LIN {X 0,Y 216.043,Z 327.914,A -85,B 0,C 180,E1 -21362.461,E2 -21362.461} C_VEL
LIN {X 0,Y 218.98,Z 315.33,A -85,B 0,C 180,E1 -21364.17,E2 -21364.17} C_VEL
LIN {X 0,Y 221.568,Z 302.387,A -85,B 0,C 180,E1 -21365.511,E2 -21365.511} C_VEL
LIN {X 0,Y 223.683,Z 288.503,A -85,B 0,C 180,E1 -21366.583,E2 -21366.583} C_VEL
LIN {X 0,Y 225.167,Z 275.245,A -85,B 0,C 180,E1 -21367.28,E2 -21367.28} C_VEL
LIN {X 0,Y 226.58,Z 250.766,A -85,B 0,C 180,E1 -21368.059,E2 -21368.059} C_VEL
LIN {X 0,Y 229.176,Z 196.259,A -85,B 0,C 180,E1 -21369.667,E2 -21369.667} C_VEL
LIN {X 0,Y 228.416,Z 191.978,A -85,B 0,C 180,E1 -21369.975,E2 -21369.975} C_VEL
LIN {X 0,Y 222.956,Z 177.944,A -85,B 0,C 180,E1 -21371.609,E2 -21371.609} C_VEL
LIN {X 0,Y 216.985,Z 164.784,A -85,B 0,C 180,E1 -21373.444,E2 -21373.444} C_VEL
LIN {X 0,Y 210.225,Z 152.018,A -85,B 0,C 180,E1 -21375.616,E2 -21375.616} C_VEL
LIN {X 0,Y 205.49,Z 143.86,A -85,B 0,C 180,E1 -21377.235,E2 -21377.235} C_VEL
LIN {X 0,Y 202.473,Z 138.962,A -85,B 0,C 180,E1 -21378.315,E2 -21378.315} C_VEL
LIN {X 0,Y 200.168,Z 135.534,A -85,B 0,C 180,E1 -21379.161,E2 -21379.161} C_VEL
LIN {X 0,Y 199.828,Z 134.46,A -85,B 0,C 180,E1 -21379.41,E2 -21379.41} C_VEL
LIN {X 0,Y 199.679,Z 133.712,A -85,B 0,C 180,E1 -21379.87,E2 -21379.87} C_VEL
LIN {X 0,Y 199.66,Z 133.735,A -85,B 0,C 180,E1 -21384.056,E2 -21384.056} C_VEL
LIN {X 0,Y 199.703,Z 133.733,A -85,B 0,C 180,E1 -21388.138,E2 -21388.138} C_VEL
LIN {X 0,Y 199.687,Z 133.735,A -85,B 0,C 180,E1 -21392.772,E2 -21392.772} C_VEL
LIN {X 0,Y 199.738,Z 133.724,A -85,B 0,C 180,E1 -21397.229,E2 -21397.229} C_VEL
LIN {X 0,Y 199.796,Z 133.708,A -85,B 0,C 180,E1 -21401.758,E2 -21401.758} C_VEL
LIN {X 0,Y 199.836,Z 133.712,A -85,B 0,C 180,E1 -21405.749,E2 -21405.749} C_VEL
LIN {X 0,Y 200.07,Z 133.686,A -85,B 0,C 180,E1 -21409.884,E2 -21409.884} C_VEL
LIN {X 0,Y 200.031,Z 133.676,A -85,B 0,C 180,E1 -21413.95,E2 -21413.95} C_VEL
LIN {X 0,Y 200.321,Z 133.658,A -85,B 0,C 180,E1 -21417.99,E2 -21417.99} C_VEL
LIN {X 0,Y 200.479,Z 133.625,A -85,B 0,C 180,E1 -21420,E2 -21420} C_VEL
LIN {X 0,Y 200.021,Z 133.683,A -85,B 0,C 180,E1 -21424.03,E2 -21424.03} C_VEL
LIN {X 0,Y 200.079,Z 133.676,A -85,B 0,C 180,E1 -21428.077,E2 -21428.077} C_VEL
LIN {X 0,Y 199.875,Z 133.703,A -85,B 0,C 180,E1 -21432.18,E2 -21432.18} C_VEL
LIN {X 0,Y 199.806,Z 133.707,A -85,B 0,C 180,E1 -21436.344,E2 -21436.344} C_VEL
LIN {X 0,Y 199.742,Z 133.728,A -85,B 0,C 180,E1 -21440.601,E2 -21440.601} C_VEL
LIN {X 0,Y 199.676,Z 133.717,A -85,B 0,C 180,E1 -21444.984,E2 -21444.984} C_VEL
LIN {X 0,Y 199.671,Z 133.734,A -85,B 0,C 180,E1 -21449.523,E2 -21449.523} C_VEL
LIN {X 0,Y 199.672,Z 133.725,A -85,B 0,C 180,E1 -21452.356,E2 -21452.356} C_VEL
LIN {X 0,Y 199.623,Z 133.732,A -85,B 0,C 180,E1 -21456.764,E2 -21456.764} C_VEL
LIN {X 0,Y 199.609,Z 133.747,A -85,B 0,C 180,E1 -21459.329,E2 -21459.329} C_VEL
LIN {X 0,Y 199.575,Z 133.74,A -85,B 0,C 180,E1 -21462.311,E2 -21462.311} C_VEL
LIN {X 0,Y 199.58,Z 133.744,A -85,B 0,C 180,E1 -21466.938,E2 -21466.938} C_VEL
LIN {X 0,Y 200.561,Z 136.528,A -85,B 0,C 180,E1 -21467.382,E2 -21467.382} C_VEL
LIN {X 0,Y 202.921,Z 139.283,A -85,B 0,C 180,E1 -21468.205,E2 -21468.205} C_VEL
LIN {X 0,Y 205.189,Z 142.628,A -85,B 0,C 180,E1 -21469,E2 -21469} C_VEL
LIN {X 0,Y 211.26,Z 151.639,A -85,B 0,C 180,E1 -21471.001,E2 -21471.001} C_VEL
LIN {X 0,Y 219.646,Z 165.612,A -85,B 0,C 180,E1 -21473.557,E2 -21473.557} C_VEL
LIN {X 0,Y 224.687,Z 176.336,A -85,B 0,C 180,E1 -21475.055,E2 -21475.055} C_VEL
LIN {X 0,Y 229.465,Z 188.114,A -85,B 0,C 180,E1 -21476.449,E2 -21476.449} C_VEL
LIN {X 0,Y 225.697,Z 264.944,A -85,B 0,C 180,E1 -21478.758,E2 -21478.758} C_VEL
LIN {X 0,Y 224.407,Z 278.641,A -85,B 0,C 180,E1 -21479.474,E2 -21479.474} C_VEL
LIN {X 0,Y 222.591,Z 291.581,A -85,B 0,C 180,E1 -21480.44,E2 -21480.44} C_VEL
LIN {X 0,Y 220.37,Z 303.982,A -85,B 0,C 180,E1 -21481.681,E2 -21481.681} C_VEL
LIN {X 0,Y 217.493,Z 316.931,A -85,B 0,C 180,E1 -21483.362,E2 -21483.362} C_VEL
LIN {X 0,Y 214.588,Z 328.651,A -85,B 0,C 180,E1 -21485.319,E2 -21485.319} C_VEL
LIN {X 0,Y 211.574,Z 339.378,A -85,B 0,C 180,E1 -21487.543,E2 -21487.543} C_VEL
LIN {X 0,Y 208.228,Z 350,A -85,B 0,C 180,E1 -21490.275,E2 -21490.275} C_VEL
LIN {X 0,Y 205.53,Z 358.756,A -85,B 0,C 180,E1 -21493.103,E2 -21493.103} C_VEL
LIN {X 0,Y 202.862,Z 367.159,A -85,B 0,C 180,E1 -21496.477,E2 -21496.477} C_VEL
LIN {X 0,Y 200.582,Z 373.941,A -85,B 0,C 180,E1 -21499.911,E2 -21499.911} C_VEL
LIN {X 0,Y 199.212,Z 378.613,A -85,B 0,C 180,E1 -21502.908,E2 -21502.908} C_VEL
LIN {X 0,Y 198.03,Z 383.462,A -85,B 0,C 180,E1 -21506.949,E2 -21506.949} C_VEL
LIN {X 0,Y 197.512,Z 386.116,A -85,B 0,C 180,E1 -21510,E2 -21510} C_VEL
LIN {X 0,Y 197.248,Z 388.443,A -85,B 0,C 180,E1 -21514.087,E2 -21514.087} C_VEL
LIN {X 0,Y 197.159,Z 389.445,A -85,B 0,C 180,E1 -21518.198,E2 -21518.198} C_VEL
LIN {X 0,Y 197.465,Z 389.126,A -85,B 0,C 180,E1 -21522.331,E2 -21522.331} C_VEL
LIN {X 0,Y 198.57,Z 387.462,A -85,B 0,C 180,E1 -21526.448,E2 -21526.448} C_VEL
LIN {X 0,Y 200.262,Z 384.414,A -85,B 0,C 180,E1 -21530.545,E2 -21530.545} C_VEL
LIN {X 0,Y 202.803,Z 379.879,A -85,B 0,C 180,E1 -21534.573,E2 -21534.573} C_VEL
LIN {X 0,Y 205.257,Z 375.362,A -85,B 0,C 180,E1 -21537.531,E2 -21537.531} C_VEL
LIN {X 0,Y 208.753,Z 368.82,A -85,B 0,C 180,E1 -21540.892,E2 -21540.892} C_VEL
LIN {X 0,Y 212.255,Z 361.917,A -85,B 0,C 180,E1 -21543.684,E2 -21543.684} C_VEL
LIN {X 0,Y 216.133,Z 353.609,A -85,B 0,C 180,E1 -21546.401,E2 -21546.401} C_VEL
LIN {X 0,Y 220.534,Z 343.57,A -85,B 0,C 180,E1 -21549.006,E2 -21549.006} C_VEL
LIN {X 0,Y 224.666,Z 333.458,A -85,B 0,C 180,E1 -21551.066,E2 -21551.066} C_VEL
LIN {X 0,Y 228.419,Z 322.488,A -85,B 0,C 180,E1 -21552.902,E2 -21552.902} C_VEL
LIN {X 0,Y 232.143,Z 310.618,A -85,B 0,C 180,E1 -21554.435,E2 -21554.435} C_VEL
LIN {X 0,Y 235.118,Z 298.588,A -85,B 0,C 180,E1 -21555.686,E2 -21555.686} C_VEL
LIN {X 0,Y 237.669,Z 285.47,A -85,B 0,C 180,E1 -21556.734,E2 -21556.734} C_VEL
LIN {X 0,Y 239.729,Z 271.443,A -85,B 0,C 180,E1 -21557.516,E2 -21557.516} C_VEL
LIN {X 0,Y 241.06,Z 256.067,A -85,B 0,C 180,E1 -21558.049,E2 -21558.049} C_VEL
LIN {X 0,Y 244.312,Z 202.285,A -85,B 0,C 180,E1 -21559.496,E2 -21559.496} C_VEL
LIN {X 0,Y 238.551,Z 189.822,A -85,B 0,C 180,E1 -21561.518,E2 -21561.518} C_VEL
LIN {X 0,Y 232.033,Z 177.432,A -85,B 0,C 180,E1 -21563.957,E2 -21563.957} C_VEL
LIN {X 0,Y 227.492,Z 170.324,A -85,B 0,C 180,E1 -21565.745,E2 -21565.745} C_VEL
LIN {X 0,Y 222.056,Z 162.557,A -85,B 0,C 180,E1 -21568.052,E2 -21568.052} C_VEL
LIN {X 0,Y 218.911,Z 158.29,A -85,B 0,C 180,E1 -21569.492,E2 -21569.492} C_VEL
LIN {X 0,Y 216.196,Z 154.622,A -85,B 0,C 180,E1 -21570.816,E2 -21570.816} C_VEL
LIN {X 0,Y 213.47,Z 151.148,A -85,B 0,C 180,E1 -21572.22,E2 -21572.22} C_VEL
LIN {X 0,Y 212.592,Z 149.965,A -85,B 0,C 180,E1 -21572.697,E2 -21572.697} C_VEL
LIN {X 0,Y 209.975,Z 147.021,A -85,B 0,C 180,E1 -21574.145,E2 -21574.145} C_VEL
LIN {X 0,Y 208.645,Z 144.909,A -85,B 0,C 180,E1 -21574.966,E2 -21574.966} C_VEL
LIN {X 0,Y 206.146,Z 142.78,A -85,B 0,C 180,E1 -21576.46,E2 -21576.46} C_VEL
LIN {X 0,Y 204.51,Z 139.754,A -85,B 0,C 180,E1 -21577.634,E2 -21577.634} C_VEL
LIN {X 0,Y 201.463,Z 137.612,A -85,B 0,C 180,E1 -21579.716,E2 -21579.716} C_VEL
LIN {X 0,Y 200.119,Z 135.295,A -85,B 0,C 180,E1 -21580.843,E2 -21580.843} C_VEL
LIN {X 0,Y 199.748,Z 133.715,A -85,B 0,C 180,E1 -21581.273,E2 -21581.273} C_VEL
LIN {X 0,Y 199.825,Z 133.705,A -85,B 0,C 180,E1 -21585.747,E2 -21585.747} C_VEL
LIN {X 0,Y 200.024,Z 133.683,A -85,B 0,C 180,E1 -21589.881,E2 -21589.881} C_VEL
LIN {X 0,Y 200.011,Z 133.696,A -85,B 0,C 180,E1 -21593.949,E2 -21593.949} C_VEL
LIN {X 0,Y 200.318,Z 133.652,A -85,B 0,C 180,E1 -21597.989,E2 -21597.989} C_VEL
LIN {X 0,Y 200.477,Z 133.626,A -85,B 0,C 180,E1 -21600,E2 -21600} C_VEL
LIN {X 0,Y 200.018,Z 133.696,A -85,B 0,C 180,E1 -21604.029,E2 -21604.029} C_VEL
LIN {X 0,Y 200.078,Z 133.68,A -85,B 0,C 180,E1 -21608.077,E2 -21608.077} C_VEL
LIN {X 0,Y 199.876,Z 133.697,A -85,B 0,C 180,E1 -21612.179,E2 -21612.179} C_VEL
LIN {X 0,Y 199.806,Z 133.703,A -85,B 0,C 180,E1 -21616.343,E2 -21616.343} C_VEL
LIN {X 0,Y 199.701,Z 133.717,A -85,B 0,C 180,E1 -21620.605,E2 -21620.605} C_VEL
LIN {X 0,Y 199.715,Z 133.82,A -85,B 0,C 180,E1 -21624.458,E2 -21624.458} C_VEL
LIN {X 0,Y 200.409,Z 136.105,A -85,B 0,C 180,E1 -21625.163,E2 -21625.163} C_VEL
LIN {X 0,Y 202.235,Z 138.346,A -85,B 0,C 180,E1 -21626.578,E2 -21626.578} C_VEL
LIN {X 0,Y 204.499,Z 139.81,A -85,B 0,C 180,E1 -21628.092,E2 -21628.092} C_VEL
LIN {X 0,Y 206.159,Z 142.761,A -85,B 0,C 180,E1 -21629.273,E2 -21629.273} C_VEL
LIN {X 0,Y 209.816,Z 146.784,A -85,B 0,C 180,E1 -21631.488,E2 -21631.488} C_VEL
LIN {X 0,Y 213.444,Z 151.85,A -85,B 0,C 180,E1 -21633.542,E2 -21633.542} C_VEL
LIN {X 0,Y 218.226,Z 158.994,A -85,B 0,C 180,E1 -21636.006,E2 -21636.006} C_VEL
LIN {X 0,Y 224.063,Z 168.172,A -85,B 0,C 180,E1 -21638.704,E2 -21638.704} C_VEL
LIN {X 0,Y 227.008,Z 173.204,A -85,B 0,C 180,E1 -21639.97,E2 -21639.97} C_VEL
LIN {X 0,Y 228.12,Z 176.401,A -85,B 0,C 180,E1 -21640.496,E2 -21640.496} C_VEL
LIN {X 0,Y 229.771,Z 189.007,A -85,B 0,C 180,E1 -21641.641,E2 -21641.641} C_VEL
LIN {X 0,Y 230.904,Z 192.261,A -85,B 0,C 180,E1 -21642.143,E2 -21642.143} C_VEL
LIN {X 0,Y 236.138,Z 203.615,A -85,B 0,C 180,E1 -21644.171,E2 -21644.171} C_VEL
LIN {X 0,Y 239.022,Z 210.694,A -85,B 0,C 180,E1 -21645.253,E2 -21645.253} C_VEL
LIN {X 0,Y 234.999,Z 272.929,A -85,B 0,C 180,E1 -21646.981,E2 -21646.981} C_VEL
LIN {X 0,Y 233.177,Z 286.688,A -85,B 0,C 180,E1 -21647.593,E2 -21647.593} C_VEL
LIN {X 0,Y 230.564,Z 300.226,A -85,B 0,C 180,E1 -21648.472,E2 -21648.472} C_VEL
LIN {X 0,Y 227.558,Z 312.525,A -85,B 0,C 180,E1 -21649.566,E2 -21649.566} C_VEL
LIN {X 0,Y 223.657,Z 325.418,A -85,B 0,C 180,E1 -21651.063,E2 -21651.063} C_VEL
LIN {X 0,Y 219.547,Z 337.241,A -85,B 0,C 180,E1 -21652.856,E2 -21652.856} C_VEL
LIN {X 0,Y 214.842,Z 349.089,A -85,B 0,C 180,E1 -21655.156,E2 -21655.156} C_VEL
LIN {X 0,Y 210.235,Z 359.289,A -85,B 0,C 180,E1 -21657.665,E2 -21657.665} C_VEL
LIN {X 0,Y 205.966,Z 367.944,A -85,B 0,C 180,E1 -21660.345,E2 -21660.345} C_VEL
LIN {X 0,Y 201.612,Z 376.267,A -85,B 0,C 180,E1 -21663.611,E2 -21663.611} C_VEL
LIN {X 0,Y 197.905,Z 382.974,A -85,B 0,C 180,E1 -21667.006,E2 -21667.006} C_VEL
LIN {X 0,Y 194.705,Z 388.95,A -85,B 0,C 180,E1 -21671.043,E2 -21671.043} C_VEL
LIN {X 0,Y 192.28,Z 393.36,A -85,B 0,C 180,E1 -21675.175,E2 -21675.175} C_VEL
LIN {X 0,Y 190.869,Z 396.345,A -85,B 0,C 180,E1 -21679.391,E2 -21679.391} C_VEL
LIN {X 0,Y 190.206,Z 397.98,A -85,B 0,C 180,E1 -21683.635,E2 -21683.635} C_VEL
LIN {X 0,Y 190.134,Z 398.292,A -85,B 0,C 180,E1 -21687.881,E2 -21687.881} C_VEL
LIN {X 0,Y 190.214,Z 397.949,A -85,B 0,C 180,E1 -21690,E2 -21690} C_VEL
LIN {X 0,Y 190.062,Z 396.762,A -85,B 0,C 180,E1 -21693.257,E2 -21693.257} C_VEL
LIN {X 0,Y 190.194,Z 394.868,A -85,B 0,C 180,E1 -21696.364,E2 -21696.364} C_VEL
LIN {X 0,Y 190.764,Z 391.039,A -85,B 0,C 180,E1 -21700.615,E2 -21700.615} C_VEL
LIN {X 0,Y 192.038,Z 385.624,A -85,B 0,C 180,E1 -21704.843,E2 -21704.843} C_VEL
LIN {X 0,Y 193.575,Z 380.437,A -85,B 0,C 180,E1 -21707.975,E2 -21707.975} C_VEL
LIN {X 0,Y 195.869,Z 372.991,A -85,B 0,C 180,E1 -21711.578,E2 -21711.578} C_VEL
LIN {X 0,Y 198.443,Z 365.185,A -85,B 0,C 180,E1 -21714.59,E2 -21714.59} C_VEL
LIN {X 0,Y 201.548,Z 355.802,A -85,B 0,C 180,E1 -21717.518,E2 -21717.518} C_VEL
LIN {X 0,Y 204.953,Z 345.411,A -85,B 0,C 180,E1 -21720.099,E2 -21720.099} C_VEL
LIN {X 0,Y 208.292,Z 333.809,A -85,B 0,C 180,E1 -21722.412,E2 -21722.412} C_VEL
LIN {X 0,Y 211.525,Z 321.198,A -85,B 0,C 180,E1 -21724.39,E2 -21724.39} C_VEL
LIN {X 0,Y 214.498,Z 307.832,A -85,B 0,C 180,E1 -21725.995,E2 -21725.995} C_VEL
LIN {X 0,Y 217.02,Z 293.84,A -85,B 0,C 180,E1 -21727.241,E2 -21727.241} C_VEL
LIN {X 0,Y 218.834,Z 280.024,A -85,B 0,C 180,E1 -21728.113,E2 -21728.113} C_VEL
LIN {X 0,Y 220.032,Z 265.889,A -85,B 0,C 180,E1 -21728.67,E2 -21728.67} C_VEL
LIN {X 0,Y 223.475,Z 197.353,A -85,B 0,C 180,E1 -21730.724,E2 -21730.724} C_VEL
LIN {X 0,Y 222.802,Z 194.105,A -85,B 0,C 180,E1 -21730.989,E2 -21730.989} C_VEL
LIN {X 0,Y 217.816,Z 181.29,A -85,B 0,C 180,E1 -21732.56,E2 -21732.56} C_VEL
LIN {X 0,Y 212.232,Z 168.773,A -85,B 0,C 180,E1 -21734.372,E2 -21734.372} C_VEL
LIN {X 0,Y 205.644,Z 156.131,A -85,B 0,C 180,E1 -21736.61,E2 -21736.61} C_VEL
LIN {X 0,Y 201.128,Z 148.295,A -85,B 0,C 180,E1 -21738.238,E2 -21738.238} C_VEL
LIN {X 0,Y 198.206,Z 143.53,A -85,B 0,C 180,E1 -21739.342,E2 -21739.342} C_VEL
LIN {X 0,Y 195.695,Z 139.581,A -85,B 0,C 180,E1 -21740.329,E2 -21740.329} C_VEL
LIN {X 0,Y 193.547,Z 137.314,A -85,B 0,C 180,E1 -21741.148,E2 -21741.148} C_VEL
LIN {X 0,Y 192.6,Z 134.586,A -85,B 0,C 180,E1 -21741.66,E2 -21741.66} C_VEL
LIN {X 0,Y 192.599,Z 134.609,A -85,B 0,C 180,E1 -21746.815,E2 -21746.815} C_VEL
LIN {X 0,Y 192.664,Z 134.603,A -85,B 0,C 180,E1 -21751.692,E2 -21751.692} C_VEL
LIN {X 0,Y 192.705,Z 134.594,A -85,B 0,C 180,E1 -21756.349,E2 -21756.349} C_VEL
LIN {X 0,Y 192.731,Z 134.587,A -85,B 0,C 180,E1 -21761.458,E2 -21761.458} C_VEL
LIN {X 0,Y 192.764,Z 134.596,A -85,B 0,C 180,E1 -21765.214,E2 -21765.214} C_VEL
LIN {X 0,Y 192.98,Z 134.566,A -85,B 0,C 180,E1 -21769.509,E2 -21769.509} C_VEL
LIN {X 0,Y 193.058,Z 134.561,A -85,B 0,C 180,E1 -21771.627,E2 -21771.627} C_VEL
LIN {X 0,Y 193.263,Z 134.537,A -85,B 0,C 180,E1 -21777.916,E2 -21777.916} C_VEL
LIN {X 0,Y 193.443,Z 134.501,A -85,B 0,C 180,E1 -21780,E2 -21780} C_VEL
LIN {X 0,Y 192.966,Z 134.563,A -85,B 0,C 180,E1 -21784.178,E2 -21784.178} C_VEL
LIN {X 0,Y 193.028,Z 134.551,A -85,B 0,C 180,E1 -21788.375,E2 -21788.375} C_VEL
LIN {X 0,Y 192.802,Z 134.588,A -85,B 0,C 180,E1 -21792.634,E2 -21792.634} C_VEL
LIN {X 0,Y 192.771,Z 134.577,A -85,B 0,C 180,E1 -21796.958,E2 -21796.958} C_VEL
LIN {X 0,Y 192.668,Z 134.611,A -85,B 0,C 180,E1 -21801.394,E2 -21801.394} C_VEL
LIN {X 0,Y 192.669,Z 134.591,A -85,B 0,C 180,E1 -21804.228,E2 -21804.228} C_VEL
LIN {X 0,Y 192.649,Z 134.614,A -85,B 0,C 180,E1 -21808.892,E2 -21808.892} C_VEL
LIN {X 0,Y 192.597,Z 134.613,A -85,B 0,C 180,E1 -21813.187,E2 -21813.187} C_VEL
LIN {X 0,Y 192.552,Z 134.618,A -85,B 0,C 180,E1 -21818.352,E2 -21818.352} C_VEL
LIN {X 0,Y 192.514,Z 134.624,A -85,B 0,C 180,E1 -21823.103,E2 -21823.103} C_VEL
LIN {X 0,Y 192.532,Z 134.623,A -85,B 0,C 180,E1 -21824.717,E2 -21824.717} C_VEL
LIN {X 0,Y 193.535,Z 137.442,A -85,B 0,C 180,E1 -21825.231,E2 -21825.231} C_VEL
LIN {X 0,Y 195.661,Z 139.673,A -85,B 0,C 180,E1 -21826.041,E2 -21826.041} C_VEL
LIN {X 0,Y 198.147,Z 143.54,A -85,B 0,C 180,E1 -21827.016,E2 -21827.016} C_VEL
LIN {X 0,Y 199.387,Z 145.114,A -85,B 0,C 180,E1 -21827.469,E2 -21827.469} C_VEL
LIN {X 0,Y 205.522,Z 154.184,A -85,B 0,C 180,E1 -21829.643,E2 -21829.643} C_VEL
LIN {X 0,Y 212.478,Z 165.472,A -85,B 0,C 180,E1 -21831.916,E2 -21831.916} C_VEL
LIN {X 0,Y 216.623,Z 173.124,A -85,B 0,C 180,E1 -21833.206,E2 -21833.206} C_VEL
LIN {X 0,Y 222.77,Z 187.419,A -85,B 0,C 180,E1 -21835.111,E2 -21835.111} C_VEL
LIN {X 0,Y 223.831,Z 190.558,A -85,B 0,C 180,E1 -21835.451,E2 -21835.451} C_VEL
LIN {X 0,Y 219.911,Z 264.951,A -85,B 0,C 180,E1 -21837.704,E2 -21837.704} C_VEL
LIN {X 0,Y 218.582,Z 278.699,A -85,B 0,C 180,E1 -21838.434,E2 -21838.434} C_VEL
LIN {X 0,Y 216.689,Z 291.669,A -85,B 0,C 180,E1 -21839.416,E2 -21839.416} C_VEL
LIN {X 0,Y 214.181,Z 304.967,A -85,B 0,C 180,E1 -21840.785,E2 -21840.785} C_VEL
LIN {X 0,Y 211.213,Z 317.757,A -85,B 0,C 180,E1 -21842.505,E2 -21842.505} C_VEL
LIN {X 0,Y 207.869,Z 330.526,A -85,B 0,C 180,E1 -21844.733,E2 -21844.733} C_VEL
LIN {X 0,Y 204.449,Z 341.937,A -85,B 0,C 180,E1 -21847.25,E2 -21847.25} C_VEL
LIN {X 0,Y 201.081,Z 352.143,A -85,B 0,C 180,E1 -21850.076,E2 -21850.076} C_VEL
LIN {X 0,Y 198.303,Z 360.573,A -85,B 0,C 180,E1 -21853,E2 -21853} C_VEL
LIN {X 0,Y 195.594,Z 368.634,A -85,B 0,C 180,E1 -21856.494,E2 -21856.494} C_VEL
LIN {X 0,Y 193.617,Z 374.316,A -85,B 0,C 180,E1 -21859.544,E2 -21859.544} C_VEL
LIN {X 0,Y 192.2,Z 378.942,A -85,B 0,C 180,E1 -21862.647,E2 -21862.647} C_VEL
LIN {X 0,Y 190.972,Z 383.749,A -85,B 0,C 180,E1 -21866.836,E2 -21866.836} C_VEL
LIN {X 0,Y 190.425,Z 386.364,A -85,B 0,C 180,E1 -21870,E2 -21870} C_VEL
LIN {X 0,Y 190.138,Z 388.653,A -85,B 0,C 180,E1 -21874.24,E2 -21874.24} C_VEL
LIN {X 0,Y 190.079,Z 389.619,A -85,B 0,C 180,E1 -21878.505,E2 -21878.505} C_VEL
LIN {X 0,Y 190.454,Z 389.262,A -85,B 0,C 180,E1 -21882.792,E2 -21882.792} C_VEL
LIN {X 0,Y 191.659,Z 387.56,A -85,B 0,C 180,E1 -21887.059,E2 -21887.059} C_VEL
LIN {X 0,Y 193.497,Z 384.473,A -85,B 0,C 180,E1 -21891.298,E2 -21891.298} C_VEL
LIN {X 0,Y 196.232,Z 379.879,A -85,B 0,C 180,E1 -21895.454,E2 -21895.454} C_VEL
LIN {X 0,Y 198.848,Z 375.333,A -85,B 0,C 180,E1 -21898.499,E2 -21898.499} C_VEL
LIN {X 0,Y 202.574,Z 368.746,A -85,B 0,C 180,E1 -21901.943,E2 -21901.943} C_VEL
LIN {X 0,Y 206.911,Z 360.53,A -85,B 0,C 180,E1 -21905.27,E2 -21905.27} C_VEL
LIN {X 0,Y 211.097,Z 351.896,A -85,B 0,C 180,E1 -21908.019,E2 -21908.019} C_VEL
LIN {X 0,Y 215.795,Z 341.395,A -85,B 0,C 180,E1 -21910.644,E2 -21910.644} C_VEL
LIN {X 0,Y 220.248,Z 330.463,A -85,B 0,C 180,E1 -21912.784,E2 -21912.784} C_VEL
LIN {X 0,Y 223.636,Z 320.662,A -85,B 0,C 180,E1 -21914.366,E2 -21914.366} C_VEL
LIN {X 0,Y 227.501,Z 308.283,A -85,B 0,C 180,E1 -21915.91,E2 -21915.91} C_VEL
LIN {X 0,Y 230.633,Z 295.583,A -85,B 0,C 180,E1 -21917.16,E2 -21917.16} C_VEL
LIN {X 0,Y 233.297,Z 281.281,A -85,B 0,C 180,E1 -21918.21,E2 -21918.21} C_VEL
LIN {X 0,Y 235.142,Z 267.584,A -85,B 0,C 180,E1 -21918.887,E2 -21918.887} C_VEL
LIN {X 0,Y 236.764,Z 245.49,A -85,B 0,C 180,E1 -21919.549,E2 -21919.549} C_VEL
LIN {X 0,Y 239.333,Z 204.883,A -85,B 0,C 180,E1 -21920.647,E2 -21920.647} C_VEL
LIN {X 0,Y 234.039,Z 193.32,A -85,B 0,C 180,E1 -21922.615,E2 -21922.615} C_VEL
LIN {X 0,Y 228.398,Z 182.356,A -85,B 0,C 180,E1 -21924.845,E2 -21924.845} C_VEL
LIN {X 0,Y 222.491,Z 173.066,A -85,B 0,C 180,E1 -21927.319,E2 -21927.319} C_VEL
LIN {X 0,Y 216.123,Z 164.126,A -85,B 0,C 180,E1 -21930.27,E2 -21930.27} C_VEL
LIN {X 0,Y 213.652,Z 160.724,A -85,B 0,C 180,E1 -21931.528,E2 -21931.528} C_VEL
LIN {X 0,Y 210.646,Z 156.65,A -85,B 0,C 180,E1 -21933.162,E2 -21933.162} C_VEL
LIN {X 0,Y 207.624,Z 153.136,A -85,B 0,C 180,E1 -21934.901,E2 -21934.901} C_VEL
LIN {X 0,Y 206.488,Z 151.387,A -85,B 0,C 180,E1 -21935.626,E2 -21935.626} C_VEL
LIN {X 0,Y 203.758,Z 148.686,A -85,B 0,C 180,E1 -21937.361,E2 -21937.361} C_VEL
LIN {X 0,Y 202.271,Z 146.094,A -85,B 0,C 180,E1 -21938.469,E2 -21938.469} C_VEL
LIN {X 0,Y 199.678,Z 144.137,A -85,B 0,C 180,E1 -21940.332,E2 -21940.332} C_VEL
LIN {X 0,Y 197.976,Z 141.157,A -85,B 0,C 180,E1 -21941.837,E2 -21941.837} C_VEL
LIN {X 0,Y 197.591,Z 140.47,A -85,B 0,C 180,E1 -21942.197,E2 -21942.197} C_VEL
LIN {X 0,Y 194.777,Z 138.754,A -85,B 0,C 180,E1 -21944.701,E2 -21944.701} C_VEL
LIN {X 0,Y 193.13,Z 136.096,A -85,B 0,C 180,E1 -21946.586,E2 -21946.586} C_VEL
LIN {X 0,Y 192.81,Z 134.579,A -85,B 0,C 180,E1 -21947.233,E2 -21947.233} C_VEL
LIN {X 0,Y 193.027,Z 134.549,A -85,B 0,C 180,E1 -21951.625,E2 -21951.625} C_VEL
LIN {X 0,Y 193.259,Z 134.529,A -85,B 0,C 180,E1 -21957.916,E2 -21957.916} C_VEL
LIN {X 0,Y 193.441,Z 134.502,A -85,B 0,C 180,E1 -21960,E2 -21960} C_VEL
LIN {X 0,Y 192.963,Z 134.573,A -85,B 0,C 180,E1 -21964.177,E2 -21964.177} C_VEL
LIN {X 0,Y 193.028,Z 134.561,A -85,B 0,C 180,E1 -21968.374,E2 -21968.374} C_VEL
LIN {X 0,Y 192.803,Z 134.581,A -85,B 0,C 180,E1 -21972.633,E2 -21972.633} C_VEL
LIN {X 0,Y 192.769,Z 134.594,A -85,B 0,C 180,E1 -21978.275,E2 -21978.275} C_VEL
LIN {X 0,Y 192.776,Z 134.846,A -85,B 0,C 180,E1 -21978.614,E2 -21978.614} C_VEL
LIN {X 0,Y 193.384,Z 136.944,A -85,B 0,C 180,E1 -21979.505,E2 -21979.505} C_VEL
LIN {X 0,Y 195.26,Z 139.274,A -85,B 0,C 180,E1 -21981.511,E2 -21981.511} C_VEL
LIN {X 0,Y 197.787,Z 140.735,A -85,B 0,C 180,E1 -21983.707,E2 -21983.707} C_VEL
LIN {X 0,Y 199.239,Z 143.602,A -85,B 0,C 180,E1 -21985.042,E2 -21985.042} C_VEL
LIN {X 0,Y 201.766,Z 145.867,A -85,B 0,C 180,E1 -21986.925,E2 -21986.925} C_VEL
LIN {X 0,Y 202.551,Z 146.584,A -85,B 0,C 180,E1 -21987.473,E2 -21987.473} C_VEL
LIN {X 0,Y 204.799,Z 149.939,A -85,B 0,C 180,E1 -21989.064,E2 -21989.064} C_VEL
LIN {X 0,Y 207.673,Z 153.228,A -85,B 0,C 180,E1 -21990.859,E2 -21990.859} C_VEL
LIN {X 0,Y 211.95,Z 159.552,A -85,B 0,C 180,E1 -21993.365,E2 -21993.365} C_VEL
LIN {X 0,Y 215.311,Z 164.593,A -85,B 0,C 180,E1 -21995.15,E2 -21995.15} C_VEL
LIN {X 0,Y 220.858,Z 173.585,A -85,B 0,C 180,E1 -21997.846,E2 -21997.846} C_VEL
LIN {X 0,Y 226.041,Z 182.769,A -85,B 0,C 180,E1 -22000.14,E2 -22000.14} C_VEL
LIN {X 0,Y 230.904,Z 192.261,A -85,B 0,C 180,E1 -22002.143,E2 -22002.143} C_VEL
LIN {X 0,Y 232.194,Z 195.309,A -85,B 0,C 180,E1 -22002.671,E2 -22002.671} C_VEL
LIN {X 0,Y 233.435,Z 200.56,A -85,B 0,C 180,E1 -22003.276,E2 -22003.276} C_VEL
LIN {X 0,Y 233.992,Z 206.248,A -85,B 0,C 180,E1 -22003.696,E2 -22003.696} C_VEL
LIN {X 0,Y 233.986,Z 214.321,A -85,B 0,C 180,E1 -22004.063,E2 -22004.063} C_VEL
LIN {X 0,Y 233.522,Z 222.478,A -85,B 0,C 180,E1 -22004.305,E2 -22004.305} C_VEL
LIN {X 0,Y 230.035,Z 273.384,A -85,B 0,C 180,E1 -22005.739,E2 -22005.739} C_VEL
LIN {X 0,Y 228.028,Z 287.696,A -85,B 0,C 180,E1 -22006.4,E2 -22006.4} C_VEL
LIN {X 0,Y 225.332,Z 300.931,A -85,B 0,C 180,E1 -22007.283,E2 -22007.283} C_VEL
LIN {X 0,Y 222.235,Z 313.041,A -85,B 0,C 180,E1 -22008.386,E2 -22008.386} C_VEL
LIN {X 0,Y 218.203,Z 325.804,A -85,B 0,C 180,E1 -22009.896,E2 -22009.896} C_VEL
LIN {X 0,Y 213.979,Z 337.416,A -85,B 0,C 180,E1 -22011.688,E2 -22011.688} C_VEL
LIN {X 0,Y 209.519,Z 348.231,A -85,B 0,C 180,E1 -22013.809,E2 -22013.809} C_VEL
LIN {X 0,Y 205.067,Z 357.817,A -85,B 0,C 180,E1 -22016.157,E2 -22016.157} C_VEL
LIN {X 0,Y 200.486,Z 366.691,A -85,B 0,C 180,E1 -22018.865,E2 -22018.865} C_VEL
LIN {X 0,Y 195.848,Z 375.206,A -85,B 0,C 180,E1 -22022.192,E2 -22022.192} C_VEL
LIN {X 0,Y 192.39,Z 381.182,A -85,B 0,C 180,E1 -22025.159,E2 -22025.159} C_VEL
LIN {X 0,Y 189.542,Z 386.144,A -85,B 0,C 180,E1 -22028.235,E2 -22028.235} C_VEL
LIN {X 0,Y 186.619,Z 391.28,A -85,B 0,C 180,E1 -22032.465,E2 -22032.465} C_VEL
LIN {X 0,Y 184.51,Z 394.93,A -85,B 0,C 180,E1 -22036.788,E2 -22036.788} C_VEL
LIN {X 0,Y 183.408,Z 397.203,A -85,B 0,C 180,E1 -22041.183,E2 -22041.183} C_VEL
LIN {X 0,Y 183.032,Z 398.146,A -85,B 0,C 180,E1 -22045.595,E2 -22045.595} C_VEL
LIN {X 0,Y 183.122,Z 397.764,A -85,B 0,C 180,E1 -22050,E2 -22050} C_VEL
LIN {X 0,Y 182.987,Z 396.716,A -85,B 0,C 180,E1 -22053.053,E2 -22053.053} C_VEL
LIN {X 0,Y 183.116,Z 394.635,A -85,B 0,C 180,E1 -22056.611,E2 -22056.611} C_VEL
LIN {X 0,Y 183.76,Z 390.771,A -85,B 0,C 180,E1 -22061.024,E2 -22061.024} C_VEL
LIN {X 0,Y 184.684,Z 386.808,A -85,B 0,C 180,E1 -22064.32,E2 -22064.32} C_VEL
LIN {X 0,Y 186.17,Z 381.928,A -85,B 0,C 180,E1 -22067.578,E2 -22067.578} C_VEL
LIN {X 0,Y 188.142,Z 375.668,A -85,B 0,C 180,E1 -22070.954,E2 -22070.954} C_VEL
LIN {X 0,Y 190.997,Z 367.496,A -85,B 0,C 180,E1 -22074.453,E2 -22074.453} C_VEL
LIN {X 0,Y 194.05,Z 358.615,A -85,B 0,C 180,E1 -22077.501,E2 -22077.501} C_VEL
LIN {X 0,Y 197.799,Z 347.86,A -85,B 0,C 180,E1 -22080.418,E2 -22080.418} C_VEL
LIN {X 0,Y 201.274,Z 336.706,A -85,B 0,C 180,E1 -22082.832,E2 -22082.832} C_VEL
LIN {X 0,Y 204.511,Z 325.039,A -85,B 0,C 180,E1 -22084.842,E2 -22084.842} C_VEL
LIN {X 0,Y 207.721,Z 311.851,A -85,B 0,C 180,E1 -22086.606,E2 -22086.606} C_VEL
LIN {X 0,Y 210.295,Z 299.162,A -85,B 0,C 180,E1 -22087.885,E2 -22087.885} C_VEL
LIN {X 0,Y 212.52,Z 284.893,A -85,B 0,C 180,E1 -22088.926,E2 -22088.926} C_VEL
LIN {X 0,Y 213.924,Z 271.536,A -85,B 0,C 180,E1 -22089.582,E2 -22089.582} C_VEL
LIN {X 0,Y 217.876,Z 198.334,A -85,B 0,C 180,E1 -22091.835,E2 -22091.835} C_VEL
LIN {X 0,Y 213.591,Z 186.571,A -85,B 0,C 180,E1 -22093.277,E2 -22093.277} C_VEL
LIN {X 0,Y 207.739,Z 173.135,A -85,B 0,C 180,E1 -22095.276,E2 -22095.276} C_VEL
LIN {X 0,Y 201.403,Z 160.723,A -85,B 0,C 180,E1 -22097.546,E2 -22097.546} C_VEL
LIN {X 0,Y 196.769,Z 152.62,A -85,B 0,C 180,E1 -22099.31,E2 -22099.31} C_VEL
LIN {X 0,Y 194.315,Z 148.514,A -85,B 0,C 180,E1 -22100.293,E2 -22100.293} C_VEL
LIN {X 0,Y 191.874,Z 144.968,A -85,B 0,C 180,E1 -22101.284,E2 -22101.284} C_VEL
LIN {X 0,Y 189.507,Z 141.818,A -85,B 0,C 180,E1 -22102.272,E2 -22102.272} C_VEL
LIN {X 0,Y 188.728,Z 140.524,A -85,B 0,C 180,E1 -22102.622,E2 -22102.622} C_VEL
LIN {X 0,Y 186.556,Z 138.308,A -85,B 0,C 180,E1 -22103.544,E2 -22103.544} C_VEL
LIN {X 0,Y 185.692,Z 136.162,A -85,B 0,C 180,E1 -22103.998,E2 -22103.998} C_VEL
LIN {X 0,Y 185.561,Z 135.49,A -85,B 0,C 180,E1 -22104.136,E2 -22104.136} C_VEL
LIN {X 0,Y 185.544,Z 135.493,A -85,B 0,C 180,E1 -22107.975,E2 -22107.975} C_VEL
LIN {X 0,Y 185.581,Z 135.483,A -85,B 0,C 180,E1 -22110.576,E2 -22110.576} C_VEL
LIN {X 0,Y 185.587,Z 135.479,A -85,B 0,C 180,E1 -22115.383,E2 -22115.383} C_VEL
LIN {X 0,Y 185.607,Z 135.479,A -85,B 0,C 180,E1 -22120.076,E2 -22120.076} C_VEL
LIN {X 0,Y 185.719,Z 135.477,A -85,B 0,C 180,E1 -22124.64,E2 -22124.64} C_VEL
LIN {X 0,Y 185.923,Z 135.442,A -85,B 0,C 180,E1 -22129.36,E2 -22129.36} C_VEL
LIN {X 0,Y 185.957,Z 135.429,A -85,B 0,C 180,E1 -22133.49,E2 -22133.49} C_VEL
LIN {X 0,Y 186.207,Z 135.416,A -85,B 0,C 180,E1 -22137.837,E2 -22137.837} C_VEL
LIN {X 0,Y 186.406,Z 135.377,A -85,B 0,C 180,E1 -22140,E2 -22140} C_VEL
LIN {X 0,Y 185.913,Z 135.442,A -85,B 0,C 180,E1 -22144.336,E2 -22144.336} C_VEL
LIN {X 0,Y 185.977,Z 135.424,A -85,B 0,C 180,E1 -22148.694,E2 -22148.694} C_VEL
LIN {X 0,Y 185.729,Z 135.472,A -85,B 0,C 180,E1 -22153.123,E2 -22153.123} C_VEL
LIN {X 0,Y 185.717,Z 135.452,A -85,B 0,C 180,E1 -22157.623,E2 -22157.623} C_VEL
LIN {X 0,Y 185.617,Z 135.487,A -85,B 0,C 180,E1 -22162.249,E2 -22162.249} C_VEL
LIN {X 0,Y 185.564,Z 135.487,A -85,B 0,C 180,E1 -22167.032,E2 -22167.032} C_VEL
LIN {X 0,Y 185.579,Z 135.489,A -85,B 0,C 180,E1 -22169.494,E2 -22169.494} C_VEL
LIN {X 0,Y 185.499,Z 135.504,A -85,B 0,C 180,E1 -22174.633,E2 -22174.633} C_VEL
LIN {X 0,Y 185.505,Z 135.489,A -85,B 0,C 180,E1 -22177.314,E2 -22177.314} C_VEL
LIN {X 0,Y 185.44,Z 135.499,A -85,B 0,C 180,E1 -22182.235,E2 -22182.235} C_VEL
LIN {X 0,Y 186.259,Z 138.017,A -85,B 0,C 180,E1 -22182.703,E2 -22182.703} C_VEL
LIN {X 0,Y 188.369,Z 140.395,A -85,B 0,C 180,E1 -22183.617,E2 -22183.617} C_VEL
LIN {X 0,Y 189.219,Z 141.412,A -85,B 0,C 180,E1 -22183.978,E2 -22183.978} C_VEL
LIN {X 0,Y 191.511,Z 144.76,A -85,B 0,C 180,E1 -22184.958,E2 -22184.958} C_VEL
LIN {X 0,Y 192.758,Z 146.418,A -85,B 0,C 180,E1 -22185.464,E2 -22185.464} C_VEL
LIN {X 0,Y 198.389,Z 154.362,A -85,B 0,C 180,E1 -22187.643,E2 -22187.643} C_VEL
LIN {X 0,Y 205.418,Z 165.512,A -85,B 0,C 180,E1 -22190.151,E2 -22190.151} C_VEL
LIN {X 0,Y 211.711,Z 176.738,A -85,B 0,C 180,E1 -22192.232,E2 -22192.232} C_VEL
LIN {X 0,Y 217.695,Z 190.968,A -85,B 0,C 180,E1 -22194.195,E2 -22194.195} C_VEL
LIN {X 0,Y 218.138,Z 192.946,A -85,B 0,C 180,E1 -22194.372,E2 -22194.372} C_VEL
LIN {X 0,Y 214.201,Z 264.949,A -85,B 0,C 180,E1 -22196.592,E2 -22196.592} C_VEL
LIN {X 0,Y 212.798,Z 278.762,A -85,B 0,C 180,E1 -22197.332,E2 -22197.332} C_VEL
LIN {X 0,Y 210.86,Z 291.752,A -85,B 0,C 180,E1 -22198.336,E2 -22198.336} C_VEL
LIN {X 0,Y 208.459,Z 304.189,A -85,B 0,C 180,E1 -22199.622,E2 -22199.622} C_VEL
LIN {X 0,Y 205.355,Z 317.162,A -85,B 0,C 180,E1 -22201.372,E2 -22201.372} C_VEL
LIN {X 0,Y 202.201,Z 328.899,A -85,B 0,C 180,E1 -22203.417,E2 -22203.417} C_VEL
LIN {X 0,Y 199.225,Z 338.673,A -85,B 0,C 180,E1 -22205.512,E2 -22205.512} C_VEL
LIN {X 0,Y 195.55,Z 349.466,A -85,B 0,C 180,E1 -22208.385,E2 -22208.385} C_VEL
LIN {X 0,Y 192.459,Z 358.373,A -85,B 0,C 180,E1 -22211.366,E2 -22211.366} C_VEL
LIN {X 0,Y 189.465,Z 366.901,A -85,B 0,C 180,E1 -22214.951,E2 -22214.951} C_VEL
LIN {X 0,Y 187.341,Z 372.889,A -85,B 0,C 180,E1 -22218.093,E2 -22218.093} C_VEL
LIN {X 0,Y 185.193,Z 379.27,A -85,B 0,C 180,E1 -22222.368,E2 -22222.368} C_VEL
LIN {X 0,Y 184.119,Z 382.979,A -85,B 0,C 180,E1 -22225.622,E2 -22225.622} C_VEL
LIN {X 0,Y 183.32,Z 386.612,A -85,B 0,C 180,E1 -22230,E2 -22230} C_VEL
LIN {X 0,Y 183.033,Z 388.864,A -85,B 0,C 180,E1 -22234.405,E2 -22234.405} C_VEL
LIN {X 0,Y 182.985,Z 389.793,A -85,B 0,C 180,E1 -22238.838,E2 -22238.838} C_VEL
LIN {X 0,Y 183.459,Z 389.398,A -85,B 0,C 180,E1 -22243.289,E2 -22243.289} C_VEL
LIN {X 0,Y 184.763,Z 387.658,A -85,B 0,C 180,E1 -22247.717,E2 -22247.717} C_VEL
LIN {X 0,Y 186.775,Z 384.532,A -85,B 0,C 180,E1 -22252.104,E2 -22252.104} C_VEL
LIN {X 0,Y 189.702,Z 379.877,A -85,B 0,C 180,E1 -22256.396,E2 -22256.396} C_VEL
LIN {X 0,Y 192.508,Z 375.308,A -85,B 0,C 180,E1 -22259.529,E2 -22259.529} C_VEL
LIN {X 0,Y 196.482,Z 368.673,A -85,B 0,C 180,E1 -22263.058,E2 -22263.058} C_VEL
LIN {X 0,Y 201.103,Z 360.251,A -85,B 0,C 180,E1 -22266.506,E2 -22266.506} C_VEL
LIN {X 0,Y 205.46,Z 351.676,A -85,B 0,C 180,E1 -22269.258,E2 -22269.258} C_VEL
LIN {X 0,Y 209.539,Z 343.054,A -85,B 0,C 180,E1 -22271.485,E2 -22271.485} C_VEL
LIN {X 0,Y 214,Z 332.772,A -85,B 0,C 180,E1 -22273.604,E2 -22273.604} C_VEL
LIN {X 0,Y 218.068,Z 321.584,A -85,B 0,C 180,E1 -22275.484,E2 -22275.484} C_VEL
LIN {X 0,Y 222.074,Z 309.401,A -85,B 0,C 180,E1 -22277.041,E2 -22277.041} C_VEL
LIN {X 0,Y 225.307,Z 296.968,A -85,B 0,C 180,E1 -22278.304,E2 -22278.304} C_VEL
LIN {X 0,Y 228.049,Z 283.162,A -85,B 0,C 180,E1 -22279.359,E2 -22279.359} C_VEL
LIN {X 0,Y 230.081,Z 269.224,A -85,B 0,C 180,E1 -22280.084,E2 -22280.084} C_VEL
LIN {X 0,Y 231.596,Z 250.185,A -85,B 0,C 180,E1 -22280.697,E2 -22280.697} C_VEL
LIN {X 0,Y 234.442,Z 207.352,A -85,B 0,C 180,E1 -22281.857,E2 -22281.857} C_VEL
LIN {X 0,Y 228.078,Z 193.625,A -85,B 0,C 180,E1 -22284.387,E2 -22284.387} C_VEL
LIN {X 0,Y 223.341,Z 184.832,A -85,B 0,C 180,E1 -22286.391,E2 -22286.391} C_VEL
LIN {X 0,Y 217.094,Z 175.159,A -85,B 0,C 180,E1 -22289.226,E2 -22289.226} C_VEL
LIN {X 0,Y 211.063,Z 166.716,A -85,B 0,C 180,E1 -22292.301,E2 -22292.301} C_VEL
LIN {X 0,Y 207.543,Z 162.09,A -85,B 0,C 180,E1 -22294.303,E2 -22294.303} C_VEL
LIN {X 0,Y 204.711,Z 158.249,A -85,B 0,C 180,E1 -22296.075,E2 -22296.075} C_VEL
LIN {X 0,Y 201.339,Z 154.429,A -85,B 0,C 180,E1 -22298.347,E2 -22298.347} C_VEL
LIN {X 0,Y 200.419,Z 152.782,A -85,B 0,C 180,E1 -22299.069,E2 -22299.069} C_VEL
LIN {X 0,Y 197.776,Z 150.47,A -85,B 0,C 180,E1 -22301.079,E2 -22301.079} C_VEL
LIN {X 0,Y 195.88,Z 147.242,A -85,B 0,C 180,E1 -22302.839,E2 -22302.839} C_VEL
LIN {X 0,Y 193.069,Z 145.172,A -85,B 0,C 180,E1 -22305.507,E2 -22305.507} C_VEL
LIN {X 0,Y 191.435,Z 142.194,A -85,B 0,C 180,E1 -22307.544,E2 -22307.544} C_VEL
LIN {X 0,Y 191.063,Z 141.457,A -85,B 0,C 180,E1 -22308.058,E2 -22308.058} C_VEL
LIN {X 0,Y 187.728,Z 139.361,A -85,B 0,C 180,E1 -22313.011,E2 -22313.011} C_VEL
LIN {X 0,Y 186.388,Z 137.069,A -85,B 0,C 180,E1 -22316.487,E2 -22316.487} C_VEL
LIN {X 0,Y 186.203,Z 135.407,A -85,B 0,C 180,E1 -22317.837,E2 -22317.837} C_VEL
LIN {X 0,Y 186.405,Z 135.378,A -85,B 0,C 180,E1 -22320,E2 -22320} C_VEL
LIN {X 0,Y 185.91,Z 135.449,A -85,B 0,C 180,E1 -22324.336,E2 -22324.336} C_VEL
LIN {X 0,Y 185.971,Z 135.637,A -85,B 0,C 180,E1 -22327.327,E2 -22327.327} C_VEL
LIN {X 0,Y 187.701,Z 139.525,A -85,B 0,C 180,E1 -22332.707,E2 -22332.707} C_VEL
LIN {X 0,Y 190.627,Z 141.357,A -85,B 0,C 180,E1 -22337.154,E2 -22337.154} C_VEL
LIN {X 0,Y 191.245,Z 141.813,A -85,B 0,C 180,E1 -22337.923,E2 -22337.923} C_VEL
LIN {X 0,Y 192.392,Z 144.402,A -85,B 0,C 180,E1 -22339.471,E2 -22339.471} C_VEL
LIN {X 0,Y 194.834,Z 146.747,A -85,B 0,C 180,E1 -22341.977,E2 -22341.977} C_VEL
LIN {X 0,Y 196.078,Z 147.569,A -85,B 0,C 180,E1 -22343.081,E2 -22343.081} C_VEL
LIN {X 0,Y 197.93,Z 150.667,A -85,B 0,C 180,E1 -22344.779,E2 -22344.779} C_VEL
LIN {X 0,Y 200.606,Z 153.154,A -85,B 0,C 180,E1 -22346.811,E2 -22346.811} C_VEL
LIN {X 0,Y 203.054,Z 156.626,A -85,B 0,C 180,E1 -22348.589,E2 -22348.589} C_VEL
LIN {X 0,Y 205.465,Z 159.52,A -85,B 0,C 180,E1 -22350.158,E2 -22350.158} C_VEL
LIN {X 0,Y 209.379,Z 165.514,A -85,B 0,C 180,E1 -22352.561,E2 -22352.561} C_VEL
LIN {X 0,Y 212.553,Z 170.4,A -85,B 0,C 180,E1 -22354.33,E2 -22354.33} C_VEL
LIN {X 0,Y 218.089,Z 179.699,A -85,B 0,C 180,E1 -22357.15,E2 -22357.15} C_VEL
LIN {X 0,Y 223.061,Z 188.878,A -85,B 0,C 180,E1 -22359.455,E2 -22359.455} C_VEL
LIN {X 0,Y 227.927,Z 198.674,A -85,B 0,C 180,E1 -22361.543,E2 -22361.543} C_VEL
LIN {X 0,Y 232.671,Z 209.405,A -85,B 0,C 180,E1 -22363.467,E2 -22363.467} C_VEL
LIN {X 0,Y 234.1,Z 213.089,A -85,B 0,C 180,E1 -22364.038,E2 -22364.038} C_VEL
LIN {X 0,Y 233.522,Z 222.478,A -85,B 0,C 180,E1 -22364.305,E2 -22364.305} C_VEL
LIN {X 0,Y 232.693,Z 228.322,A -85,B 0,C 180,E1 -22364.342,E2 -22364.342} C_VEL
LIN {X 0,Y 227.626,Z 247.365,A -85,B 0,C 180,E1 -22363.794,E2 -22363.794} C_VEL
LIN {X 0,Y 226.765,Z 253.212,A -85,B 0,C 180,E1 -22363.821,E2 -22363.821} C_VEL
LIN {X 0,Y 225.044,Z 274.995,A -85,B 0,C 180,E1 -22364.488,E2 -22364.488} C_VEL
LIN {X 0,Y 222.989,Z 288.715,A -85,B 0,C 180,E1 -22365.154,E2 -22365.154} C_VEL
LIN {X 0,Y 220.2,Z 301.646,A -85,B 0,C 180,E1 -22366.038,E2 -22366.038} C_VEL
LIN {X 0,Y 217.01,Z 313.562,A -85,B 0,C 180,E1 -22367.149,E2 -22367.149} C_VEL
LIN {X 0,Y 212.839,Z 326.194,A -85,B 0,C 180,E1 -22368.669,E2 -22368.669} C_VEL
LIN {X 0,Y 208.472,Z 337.705,A -85,B 0,C 180,E1 -22370.482,E2 -22370.482} C_VEL
LIN {X 0,Y 203.623,Z 348.907,A -85,B 0,C 180,E1 -22372.734,E2 -22372.734} C_VEL
LIN {X 0,Y 198.378,Z 359.591,A -85,B 0,C 180,E1 -22375.47,E2 -22375.47} C_VEL
LIN {X 0,Y 193.72,Z 368.141,A -85,B 0,C 180,E1 -22378.261,E2 -22378.261} C_VEL
LIN {X 0,Y 188.95,Z 376.346,A -85,B 0,C 180,E1 -22381.69,E2 -22381.69} C_VEL
LIN {X 0,Y 184.854,Z 382.966,A -85,B 0,C 180,E1 -22385.278,E2 -22385.278} C_VEL
LIN {X 0,Y 182.099,Z 387.546,A -85,B 0,C 180,E1 -22388.491,E2 -22388.491} C_VEL
LIN {X 0,Y 179.833,Z 391.219,A -85,B 0,C 180,E1 -22391.781,E2 -22391.781} C_VEL
LIN {X 0,Y 177.553,Z 394.837,A -85,B 0,C 180,E1 -22396.261,E2 -22396.261} C_VEL
LIN {X 0,Y 176.355,Z 397.078,A -85,B 0,C 180,E1 -22400.827,E2 -22400.827} C_VEL
LIN {X 0,Y 175.944,Z 397.99,A -85,B 0,C 180,E1 -22405.417,E2 -22405.417} C_VEL
LIN {X 0,Y 176.031,Z 397.578,A -85,B 0,C 180,E1 -22410,E2 -22410} C_VEL
LIN {X 0,Y 175.933,Z 395.806,A -85,B 0,C 180,E1 -22414.582,E2 -22414.582} C_VEL
LIN {X 0,Y 176.317,Z 392.64,A -85,B 0,C 180,E1 -22419.174,E2 -22419.174} C_VEL
LIN {X 0,Y 177.321,Z 387.945,A -85,B 0,C 180,E1 -22423.757,E2 -22423.757} C_VEL
LIN {X 0,Y 178.79,Z 383.354,A -85,B 0,C 180,E1 -22427.146,E2 -22427.146} C_VEL
LIN {X 0,Y 180.654,Z 377.725,A -85,B 0,C 180,E1 -22430.495,E2 -22430.495} C_VEL
LIN {X 0,Y 183.517,Z 369.704,A -85,B 0,C 180,E1 -22434.31,E2 -22434.31} C_VEL
LIN {X 0,Y 186.599,Z 361.309,A -85,B 0,C 180,E1 -22437.476,E2 -22437.476} C_VEL
LIN {X 0,Y 190.313,Z 351.197,A -85,B 0,C 180,E1 -22440.515,E2 -22440.515} C_VEL
LIN {X 0,Y 193.737,Z 341.008,A -85,B 0,C 180,E1 -22442.965,E2 -22442.965} C_VEL
LIN {X 0,Y 197.088,Z 329.984,A -85,B 0,C 180,E1 -22445.099,E2 -22445.099} C_VEL
LIN {X 0,Y 200.331,Z 318.046,A -85,B 0,C 180,E1 -22446.925,E2 -22446.925} C_VEL
LIN {X 0,Y 203.401,Z 304.944,A -85,B 0,C 180,E1 -22448.458,E2 -22448.458} C_VEL
LIN {X 0,Y 205.969,Z 290.601,A -85,B 0,C 180,E1 -22449.695,E2 -22449.695} C_VEL
LIN {X 0,Y 207.819,Z 276.217,A -85,B 0,C 180,E1 -22450.543,E2 -22450.543} C_VEL
LIN {X 0,Y 209.182,Z 257.283,A -85,B 0,C 180,E1 -22451.209,E2 -22451.209} C_VEL
LIN {X 0,Y 212.347,Z 200.076,A -85,B 0,C 180,E1 -22452.975,E2 -22452.975} C_VEL
LIN {X 0,Y 207.238,Z 186.627,A -85,B 0,C 180,E1 -22454.783,E2 -22454.783} C_VEL
LIN {X 0,Y 201.846,Z 174.412,A -85,B 0,C 180,E1 -22456.756,E2 -22456.756} C_VEL
LIN {X 0,Y 195.911,Z 162.932,A -85,B 0,C 180,E1 -22459.036,E2 -22459.036} C_VEL
LIN {X 0,Y 190.75,Z 153.94,A -85,B 0,C 180,E1 -22461.165,E2 -22461.165} C_VEL
LIN {X 0,Y 188.096,Z 150.142,A -85,B 0,C 180,E1 -22462.294,E2 -22462.294} C_VEL
LIN {X 0,Y 185.16,Z 146.12,A -85,B 0,C 180,E1 -22463.601,E2 -22463.601} C_VEL
LIN {X 0,Y 182.795,Z 143.054,A -85,B 0,C 180,E1 -22464.702,E2 -22464.702} C_VEL
LIN {X 0,Y 181.929,Z 141.616,A -85,B 0,C 180,E1 -22465.139,E2 -22465.139} C_VEL
LIN {X 0,Y 179.64,Z 139.458,A -85,B 0,C 180,E1 -22466.229,E2 -22466.229} C_VEL
LIN {X 0,Y 178.621,Z 137.054,A -85,B 0,C 180,E1 -22466.828,E2 -22466.828} C_VEL
LIN {X 0,Y 178.5,Z 136.365,A -85,B 0,C 180,E1 -22467.055,E2 -22467.055} C_VEL
